KUKA KRL program: MyProgram_270().src

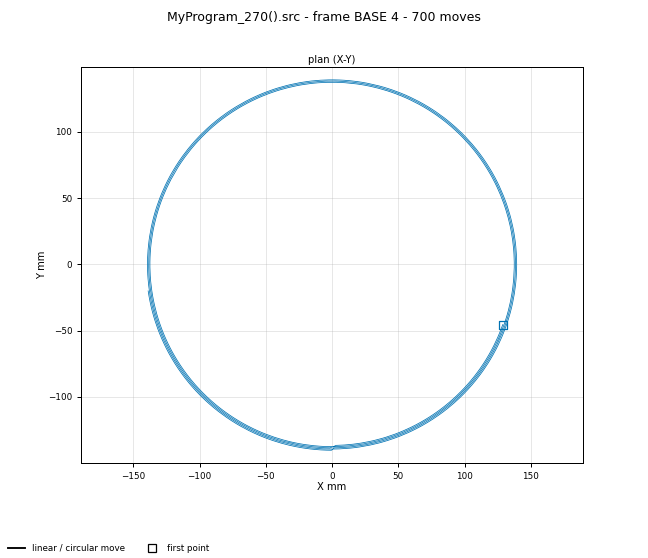
[picture p0: tool path of MyProgram_270().src in frame BASE 4, 700 of 700 moves have a stored position in this frame; points joined in program order, loops and branches not executed]
&ACCESS RVP
&REL 1
&PARAM TEMPLATE = C:\KRC\Roboter\Template\vorgabe
&PARAM EDITMASK = *
DEF MyProgram_270()
; ---- Setting reference (Base) ----
$BASE = BASE_DATA[4]

; --------------------------
; ---- Setting tool (TCP) ----
$TOOL = TOOL_DATA[3]
; --------------------------

$VEL.CP = VEL_APROX_PRINT
Startdeposition()
$VEL.CP = VEL_PRINT
LIN {X 128.8267,Y -45.3786,Z 170,A -18.166,B 9.5893,C 0.2653,E1 9.7435,E2 469.4247} C_DIS
LIN {X 127.6673,Y -48.5446,Z 170,A -19.5524,B 9.5893,C 0.2686,E1 9.7422,E2 470.8092} C_DIS
LIN {X 126.4689,Y -51.5847,Z 170,A -20.9292,B 9.5891,C 0.2724,E1 9.7407,E2 472.1882} C_DIS
LIN {X 125.0288,Y -54.9869,Z 170,A -22.4429,B 9.5891,C 0.2758,E1 9.7391,E2 473.6991} C_DIS
LIN {X 123.6815,Y -57.9517,Z 170,A -23.7911,B 9.589,C 0.2791,E1 9.7375,E2 475.0465} C_DIS
LIN {X 122.1838,Y -61.0461,Z 170,A -25.2077,B 9.5889,C 0.2823,E1 9.7358,E2 476.4613} C_DIS
LIN {X 120.4787,Y -64.3474,Z 170,A -26.8785,B 9.5887,C 0.289,E1 9.7336,E2 478.148} C_DIS
LIN {X 118.4664,Y -67.9811,Z 170,A -28.5284,B 9.5886,C 0.2914,E1 9.7313,E2 479.7881} C_DIS
LIN {X 116.2405,Y -71.7206,Z 170,A -30.2842,B 9.5885,C 0.2944,E1 9.7288,E2 481.5371} C_DIS
LIN {X 114.1692,Y -74.9733,Z 170,A -31.9695,B 9.5883,C 0.3,E1 9.7262,E2 483.2326} C_DIS
LIN {X 111.5417,Y -78.8293,Z 170,A -33.8376,B 9.5883,C 0.3027,E1 9.7233,E2 485.0916} C_DIS
LIN {X 109.2893,Y -81.9245,Z 170,A -35.3836,B 9.5882,C 0.3052,E1 9.7207,E2 486.6318} C_DIS
LIN {X 107.1942,Y -84.647,Z 170,A -36.8457,B 9.588,C 0.3091,E1 9.7182,E2 488.098} C_DIS
LIN {X 104.5097,Y -87.9395,Z 170,A -38.5977,B 9.588,C 0.3125,E1 9.7151,E2 489.8481} C_DIS
LIN {X 102.0952,Y -90.7319,Z 170,A -40.1071,B 9.5878,C 0.3151,E1 9.7123,E2 491.3542} C_DIS
LIN {X 99.655,Y -93.4058,Z 170,A -41.5996,B 9.5878,C 0.3179,E1 9.7095,E2 492.8449} C_DIS
LIN {X 97.2867,Y -95.8696,Z 170,A -43.1095,B 9.5876,C 0.3227,E1 9.7065,E2 494.3659} C_DIS
LIN {X 94.0487,Y -99.0485,Z 170,A -44.8992,B 9.5876,C 0.3241,E1 9.703,E2 496.1433} C_DIS
LIN {X 91.4543,Y -101.4489,Z 170,A -46.374,B 9.5875,C 0.327,E1 9.6999,E2 497.6185} C_DIS
LIN {X 88.8005,Y -103.7798,Z 170,A -47.8905,B 9.5873,C 0.3307,E1 9.6967,E2 499.1409} C_DIS
LIN {X 85.4707,Y -106.5386,Z 170,A -49.6437,B 9.5873,C 0.3328,E1 9.6929,E2 500.8882} C_DIS
LIN {X 82.6267,Y -108.7594,Z 170,A -51.1246,B 9.5872,C 0.3349,E1 9.6896,E2 502.3665} C_DIS
LIN {X 79.7996,Y -110.8504,Z 170,A -52.6158,B 9.5871,C 0.338,E1 9.6863,E2 503.8611} C_DIS
LIN {X 76.3701,Y -113.2397,Z 170,A -54.3449,B 9.587,C 0.3405,E1 9.6823,E2 505.5887} C_DIS
LIN {X 73.3437,Y -115.2233,Z 170,A -55.8332,B 9.587,C 0.3424,E1 9.6788,E2 507.0747} C_DIS
LIN {X 70.377,Y -117.0589,Z 170,A -57.2831,B 9.5868,C 0.3444,E1 9.6754,E2 508.5243} C_DIS
LIN {X 67.0538,Y -118.9933,Z 170,A -58.9763,B 9.5867,C 0.3487,E1 9.6712,E2 510.229} C_DIS
LIN {X 63.1615,Y -121.1024,Z 170,A -60.7503,B 9.5867,C 0.3496,E1 9.6669,E2 511.994} C_DIS
LIN {X 59.6528,Y -122.8711,Z 170,A -62.3575,B 9.5867,C 0.351,E1 9.6629,E2 513.5976} C_DIS
LIN {X 56.5477,Y -124.3307,Z 170,A -63.7852,B 9.5866,C 0.3527,E1 9.6593,E2 515.025} C_DIS
LIN {X 53.8192,Y -125.5337,Z 170,A -65.022,B 9.5866,C 0.3539,E1 9.6561,E2 516.2609} C_DIS
LIN {X 50.4299,Y -126.9344,Z 170,A -66.5584,B 9.5864,C 0.3557,E1 9.6521,E2 517.7984} C_DIS
LIN {X 47.1173,Y -128.2019,Z 170,A -68.0301,B 9.5864,C 0.3571,E1 9.6483,E2 519.2693} C_DIS
LIN {X 43.9464,Y -129.3232,Z 170,A -69.4316,B 9.5864,C 0.3584,E1 9.6446,E2 520.6707} C_DIS
LIN {X 40.9221,Y -130.3108,Z 170,A -70.7407,B 9.5864,C 0.3592,E1 9.6411,E2 521.9775} C_DIS
LIN {X 37.7424,Y -131.267,Z 170,A -72.1466,B 9.5863,C 0.3608,E1 9.6373,E2 523.3861} C_DIS
LIN {X 34.3963,Y -132.1842,Z 170,A -73.588,B 9.5863,C 0.3617,E1 9.6334,E2 524.8268} C_DIS
LIN {X 31.6889,Y -132.8572,Z 170,A -74.7716,B 9.5862,C 0.363,E1 9.6302,E2 526.0128} C_DIS
LIN {X 28.5021,Y -133.5771,Z 170,A -76.1439,B 9.5862,C 0.364,E1 9.6265,E2 527.3863} C_DIS
LIN {X 24.8536,Y -134.3059,Z 170,A -77.6673,B 9.5862,C 0.3643,E1 9.6223,E2 528.906} C_DIS
LIN {X 21.8419,Y -134.8276,Z 170,A -78.9427,B 9.5861,C 0.3649,E1 9.6188,E2 530.1813} C_DIS
LIN {X 18.6875,Y -135.3009,Z 170,A -80.275,B 9.5861,C 0.3655,E1 9.6151,E2 531.5137} C_DIS
LIN {X 15.9333,Y -135.6516,Z 170,A -81.4857,B 9.5861,C 0.367,E1 9.6117,E2 532.7309} C_DIS
LIN {X 12.4247,Y -136.0191,Z 170,A -82.9083,B 9.5861,C 0.3664,E1 9.6078,E2 534.1471} C_DIS
LIN {X 9.1702,Y -136.278,Z 170,A -84.2729,B 9.5861,C 0.3668,E1 9.604,E2 535.5119} C_DIS
LIN {X 6.089,Y -136.4504,Z 170,A -85.5634,B 9.5861,C 0.3671,E1 9.6004,E2 536.8026} C_DIS
LIN {X 3.0317,Y -136.5525,Z 170,A -86.8425,B 9.5861,C 0.3672,E1 9.5968,E2 538.0818} C_DIS
LIN {X 3.0317,Y -136.5525,Z 170,A -86.8425,B 9.5861,C 0.3672,E1 9.5968,E2 538.0818} C_DIS
Enddeposition()
LIN {X 0.9945,Y -137.4915,Z 170,A -87.085,B 9.5192,C 0.3619,E1 9.5293,E2 538.3005} C_DIS
Startdeposition()
$VEL.CP = VEL_PRINT
LIN {X 4.4577,Y -137.425,Z 170,A -85.4345,B 9.5194,C 0.3572,E1 9.534,E2 536.6227} C_DIS
LIN {X 8.6389,Y -137.2242,Z 170,A -83.302,B 9.5198,C 0.3482,E1 9.5401,E2 534.4389} C_DIS
LIN {X 13.382,Y -136.8431,Z 170,A -81.8432,B 9.5194,C 0.3589,E1 9.5439,E2 533.0469} C_DIS
LIN {X 19.4211,Y -136.1171,Z 170,A -79.3116,B 9.5194,C 0.3577,E1 9.5509,E2 530.5142} C_DIS
LIN {X 23.2629,Y -135.5149,Z 170,A -77.6681,B 9.5194,C 0.3562,E1 9.5555,E2 528.8668} C_DIS
LIN {X 27.2986,Y -134.7584,Z 170,A -76.0431,B 9.5194,C 0.3569,E1 9.5599,E2 527.2517} C_DIS
LIN {X 30.5689,Y -134.0543,Z 170,A -74.6502,B 9.5194,C 0.3559,E1 9.5637,E2 525.8579} C_DIS
LIN {X 34.5877,Y -133.0763,Z 170,A -72.9496,B 9.5195,C 0.355,E1 9.5683,E2 524.1592} C_DIS
LIN {X 38.9693,Y -131.8579,Z 170,A -71.0112,B 9.5196,C 0.3523,E1 9.5735,E2 522.2138} C_DIS
LIN {X 45.6098,Y -129.7115,Z 170,A -68.1707,B 9.5196,C 0.3508,E1 9.5811,E2 519.3799} C_DIS
LIN {X 50.1018,Y -128.0424,Z 170,A -66.1842,B 9.5197,C 0.3488,E1 9.5862,E2 517.3932} C_DIS
LIN {X 53.7419,Y -126.56,Z 170,A -64.1199,B 9.5201,C 0.3371,E1 9.5917,E2 515.2725} C_DIS
LIN {X 57.296,Y -124.9893,Z 170,A -63.0785,B 9.5198,C 0.3481,E1 9.5942,E2 514.3044} C_DIS
LIN {X 59.6774,Y -123.8699,Z 170,A -61.8597,B 9.5199,C 0.3438,E1 9.5973,E2 513.0689} C_DIS
LIN {X 62.703,Y -122.3658,Z 170,A -60.4224,B 9.52,C 0.3411,E1 9.6009,E2 511.6267} C_DIS
LIN {X 66.3461,Y -120.4316,Z 170,A -58.5872,B 9.5202,C 0.3359,E1 9.6054,E2 509.7749} C_DIS
LIN {X 70.6496,Y -117.9585,Z 170,A -56.733,B 9.5202,C 0.3376,E1 9.6098,E2 507.9465} C_DIS
LIN {X 72.7662,Y -116.6644,Z 170,A -55.6329,B 9.5202,C 0.3344,E1 9.6125,E2 506.837} C_DIS
LIN {X 76.2614,Y -114.4102,Z 170,A -53.8574,B 9.5204,C 0.3305,E1 9.6166,E2 505.0544} C_DIS
LIN {X 80.3711,Y -111.5619,Z 170,A -51.3205,B 9.5209,C 0.3162,E1 9.6225,E2 502.4569} C_DIS
LIN {X 84.1974,Y -108.7027,Z 170,A -49.8119,B 9.5206,C 0.3237,E1 9.6257,E2 501.0088} C_DIS
LIN {X 87.6291,Y -105.9558,Z 170,A -47.4584,B 9.5211,C 0.308,E1 9.631,E2 498.5859} C_DIS
LIN {X 91.5947,Y -102.5472,Z 170,A -46.0081,B 9.5207,C 0.3207,E1 9.6338,E2 497.2277} C_DIS
LIN {X 96.5572,Y -97.8895,Z 170,A -43.2267,B 9.5209,C 0.3161,E1 9.6394,E2 494.4507} C_DIS
LIN {X 101.1452,Y -93.1405,Z 170,A -40.3451,B 9.5212,C 0.307,E1 9.645,E2 491.5496} C_DIS
LIN {X 103.3355,Y -90.7051,Z 170,A -38.9793,B 9.5212,C 0.3039,E1 9.6476,E2 490.1823} C_DIS
LIN {X 106.1515,Y -87.3928,Z 170,A -37.1754,B 9.5214,C 0.2999,E1 9.6508,E2 488.3775} C_DIS
LIN {X 109.5395,Y -83.1066,Z 170,A -35.0798,B 9.5214,C 0.2989,E1 9.6543,E2 486.3028} C_DIS
LIN {X 111.5125,Y -80.4397,Z 170,A -33.6162,B 9.5216,C 0.2936,E1 9.6568,E2 484.8273} C_DIS
LIN {X 113.8575,Y -77.0841,Z 170,A -31.9629,B 9.5216,C 0.2906,E1 9.6594,E2 483.179} C_DIS
LIN {X 117.9408,Y -70.6793,Z 170,A -29.0515,B 9.5217,C 0.2888,E1 9.6637,E2 480.2969} C_DIS
LIN {X 120.0387,Y -67.0547,Z 170,A -27.0708,B 9.522,C 0.2786,E1 9.6665,E2 478.2841} C_DIS
LIN {X 122.0959,Y -63.2308,Z 170,A -25.3145,B 9.5221,C 0.2751,E1 9.6687,E2 476.5327} C_DIS
LIN {X 124.9836,Y -57.3082,Z 170,A -22.6476,B 9.5223,C 0.2697,E1 9.672,E2 473.8731} C_DIS
LIN {X 126.4048,Y -54.102,Z 170,A -21.2081,B 9.5223,C 0.2663,E1 9.6736,E2 472.4348} C_DIS
LIN {X 127.992,Y -50.2314,Z 170,A -19.2693,B 9.5226,C 0.2568,E1 9.6756,E2 470.469} C_DIS
LIN {X 129.8776,Y -45.1308,Z 170,A -17.2435,B 9.5226,C 0.2563,E1 9.6775,E2 468.4716} C_DIS
LIN {X 131.0142,Y -41.7167,Z 170,A -15.7755,B 9.5227,C 0.2529,E1 9.6788,E2 467.006} C_DIS
LIN {X 132.121,Y -38.0707,Z 170,A -14.1922,B 9.5228,C 0.2485,E1 9.68,E2 465.4217} C_DIS
LIN {X 133.0849,Y -34.5541,Z 170,A -12.7534,B 9.5229,C 0.2461,E1 9.681,E2 463.9916} C_DIS
LIN {X 133.941,Y -31.065,Z 170,A -11.3472,B 9.5229,C 0.244,E1 9.682,E2 462.5954} C_DIS
LIN {X 134.5739,Y -28.2049,Z 170,A -9.7939,B 9.5232,C 0.2325,E1 9.6829,E2 460.9984} C_DIS
LIN {X 135.7493,Y -21.8581,Z 170,A -7.1388,B 9.5234,C 0.2256,E1 9.6841,E2 458.3449} C_DIS
LIN {X 136.3722,Y -17.5435,Z 170,A -5.5976,B 9.5234,C 0.227,E1 9.6847,E2 456.8371} C_DIS
LIN {X 137.0353,Y -11.2466,Z 170,A -3.001,B 9.5235,C 0.2203,E1 9.6854,E2 454.2432} C_DIS
LIN {X 137.4746,Y -2.4202,Z 170,A 0.3604,B 9.5236,C 0.2174,E1 9.6859,E2 450.9192} C_DIS
LIN {X 137.4858,Y 1.6825,Z 170,A 2.4979,B 9.5239,C 0.2021,E1 9.6859,E2 448.7258} C_DIS
LIN {X 137.2829,Y 7.638,Z 170,A 5.1259,B 9.5242,C 0.1914,E1 9.6855,E2 446.077} C_DIS
LIN {X 137.0196,Y 11.4331,Z 170,A 6.7511,B 9.5242,C 0.1858,E1 9.6851,E2 444.4452} C_DIS
LIN {X 136.6061,Y 15.6289,Z 170,A 7.9732,B 9.5242,C 0.1937,E1 9.6848,E2 443.2897} C_DIS
LIN {X 136.2687,Y 18.3336,Z 170,A 9.3236,B 9.5242,C 0.1852,E1 9.6842,E2 441.911} C_DIS
LIN {X 135.7575,Y 21.8067,Z 170,A 10.5805,B 9.5242,C 0.186,E1 9.6837,E2 440.679} C_DIS
LIN {X 135.2539,Y 24.7321,Z 170,A 11.8194,B 9.5243,C 0.1824,E1 9.6831,E2 439.4387} C_DIS
LIN {X 134.373,Y 29.1363,Z 170,A 13.5842,B 9.5243,C 0.1796,E1 9.6821,E2 437.6859} C_DIS
LIN {X 133.6464,Y 32.3057,Z 170,A 14.9678,B 9.5245,C 0.1751,E1 9.6812,E2 436.2976} C_DIS
LIN {X 132.816,Y 35.5659,Z 170,A 16.385,B 9.5245,C 0.1708,E1 9.6802,E2 434.8773} C_DIS
LIN {X 131.8736,Y 38.9155,Z 170,A 17.7516,B 9.5245,C 0.1688,E1 9.6792,E2 433.52} C_DIS
LIN {X 130.8981,Y 42.0801,Z 170,A 19.18,B 9.5247,C 0.1638,E1 9.678,E2 432.0845} C_DIS
LIN {X 129.6333,Y 45.8355,Z 170,A 21.2102,B 9.5249,C 0.1503,E1 9.6761,E2 430.0051} C_DIS
LIN {X 128.3016,Y 49.435,Z 170,A 22.2113,B 9.5247,C 0.1602,E1 9.6752,E2 429.0785} C_DIS
LIN {X 127.125,Y 52.3889,Z 170,A 23.6027,B 9.5248,C 0.1551,E1 9.6737,E2 427.6778} C_DIS
LIN {X 126.162,Y 54.6637,Z 170,A 24.7189,B 9.5248,C 0.1503,E1 9.6724,E2 426.5499} C_DIS
LIN {X 124.6519,Y 58.0255,Z 170,A 26.237,B 9.5249,C 0.1467,E1 9.6707,E2 425.033} C_DIS
LIN {X 123.119,Y 61.2114,Z 170,A 27.7436,B 9.525,C 0.1421,E1 9.6688,E2 423.5213} C_DIS
LIN {X 120.9378,Y 65.4193,Z 170,A 29.7086,B 9.525,C 0.1373,E1 9.6662,E2 421.5563} C_DIS
LIN {X 118.8946,Y 69.0623,Z 170,A 31.4905,B 9.5252,C 0.132,E1 9.6638,E2 419.7682} C_DIS
LIN {X 116.9053,Y 72.3792,Z 170,A 32.9669,B 9.5252,C 0.1312,E1 9.6616,E2 418.3078} C_DIS
LIN {X 114.6044,Y 75.9704,Z 170,A 34.7336,B 9.5252,C 0.1271,E1 9.6589,E2 416.5416} C_DIS
LIN {X 112.1602,Y 79.5342,Z 170,A 36.5435,B 9.5252,C 0.1227,E1 9.656,E2 414.7295} C_DIS
LIN {X 109.5062,Y 83.1507,Z 170,A 38.4153,B 9.5253,C 0.1183,E1 9.6529,E2 412.8565} C_DIS
LIN {X 106.7022,Y 86.7194,Z 170,A 40.289,B 9.5253,C 0.1145,E1 9.6496,E2 410.9842} C_DIS
LIN {X 103.7598,Y 90.2188,Z 170,A 42.1695,B 9.5254,C 0.1109,E1 9.6462,E2 409.106} C_DIS
LIN {X 99.0767,Y 95.3387,Z 170,A 44.8966,B 9.5254,C 0.1086,E1 9.6411,E2 406.3984} C_DIS
LIN {X 96.5488,Y 97.8977,Z 170,A 46.6566,B 9.5255,C 0.0996,E1 9.6375,E2 404.6051} C_DIS
LIN {X 93.4602,Y 100.8503,Z 170,A 48.2466,B 9.5255,C 0.1005,E1 9.6344,E2 403.0385} C_DIS
LIN {X 90.203,Y 103.7736,Z 170,A 50.0397,B 9.5255,C 0.0977,E1 9.6306,E2 401.2487} C_DIS
LIN {X 86.7906,Y 106.644,Z 170,A 51.8616,B 9.5255,C 0.0951,E1 9.6267,E2 399.4308} C_DIS
LIN {X 83.3506,Y 109.3536,Z 170,A 53.6942,B 9.5256,C 0.0918,E1 9.6226,E2 397.5968} C_DIS
LIN {X 78.9782,Y 112.5524,Z 170,A 55.7465,B 9.5256,C 0.0926,E1 9.6181,E2 395.5697} C_DIS
LIN {X 76.5732,Y 114.202,Z 170,A 57.1185,B 9.5256,C 0.0871,E1 9.6148,E2 394.178} C_DIS
LIN {X 72.947,Y 116.5519,Z 170,A 58.917,B 9.5256,C 0.0844,E1 9.6106,E2 392.3796} C_DIS
LIN {X 69.2198,Y 118.8034,Z 170,A 60.7573,B 9.5257,C 0.0812,E1 9.6062,E2 390.5359} C_DIS
LIN {X 65.4765,Y 120.907,Z 170,A 62.5302,B 9.5257,C 0.0791,E1 9.6018,E2 388.7649} C_DIS
LIN {X 60.8601,Y 123.2922,Z 170,A 64.3876,B 9.5257,C 0.0831,E1 9.5973,E2 386.9457} C_DIS
LIN {X 58.71,Y 124.332,Z 170,A 65.5408,B 9.5257,C 0.0784,E1 9.5944,E2 385.773} C_DIS
LIN {X 55.751,Y 125.6859,Z 170,A 66.8596,B 9.5257,C 0.0777,E1 9.591,E2 384.4588} C_DIS
LIN {X 52.3572,Y 127.1383,Z 170,A 68.4709,B 9.5257,C 0.0744,E1 9.5868,E2 382.8386} C_DIS
LIN {X 47.9866,Y 128.8499,Z 170,A 70.365,B 9.5257,C 0.0737,E1 9.5819,E2 380.9522} C_DIS
LIN {X 44.9262,Y 129.9485,Z 170,A 71.7246,B 9.5257,C 0.0724,E1 9.5783,E2 379.5922} C_DIS
LIN {X 41.4522,Y 131.0986,Z 170,A 73.2785,B 9.5258,C 0.0704,E1 9.5742,E2 378.0349} C_DIS
LIN {X 38.1638,Y 132.0937,Z 170,A 74.639,B 9.5258,C 0.0708,E1 9.5706,E2 376.6835} C_DIS
LIN {X 34.9179,Y 132.9888,Z 170,A 76.1705,B 9.5258,C 0.0671,E1 9.5664,E2 375.1363} C_DIS
LIN {X 29.0493,Y 134.3918,Z 170,A 78.6429,B 9.5258,C 0.0664,E1 9.5597,E2 372.6698} C_DIS
LIN {X 25.6384,Y 135.0841,Z 170,A 80.0199,B 9.5258,C 0.0672,E1 9.5559,E2 371.3023} C_DIS
LIN {X 21.8795,Y 135.7457,Z 170,A 81.9193,B 9.5258,C 0.06,E1 9.5506,E2 369.3651} C_DIS
LIN {X 18.5277,Y 136.2432,Z 170,A 83.1255,B 9.5258,C 0.0638,E1 9.5473,E2 368.1849} C_DIS
LIN {X 9.7314,Y 137.1512,Z 170,A 87.6017,B 9.5259,C 0.0464,E1 9.5346,E2 363.6113} C_DIS
LIN {X 3.0399,Y 137.4642,Z 170,A 89.441,B 9.5259,C 0.066,E1 9.5298,E2 361.892} C_DIS
LIN {X -4.0559,Y 137.4362,Z 170,A 92.5213,B 9.5259,C 0.0637,E1 9.5212,E2 358.798} C_DIS
LIN {X -10.5289,Y 137.093,Z 170,A 95.0095,B 9.5259,C 0.0686,E1 9.5143,E2 356.3376} C_DIS
LIN {X -15.8028,Y 136.5853,Z 170,A 97.2212,B 9.5259,C 0.0692,E1 9.5082,E2 354.1268} C_DIS
LIN {X -19.7314,Y 136.0727,Z 170,A 99.2909,B 9.5259,C 0.0615,E1 9.5023,E2 352.0062} C_DIS
LIN {X -22.8961,Y 135.5761,Z 170,A 100.445,B 9.5259,C 0.0658,E1 9.4992,E2 350.8753} C_DIS
LIN {X -26.4326,Y 134.9321,Z 170,A 101.8121,B 9.5259,C 0.0693,E1 9.4955,E2 349.5254} C_DIS
LIN {X -30.0751,Y 134.1671,Z 170,A 103.299,B 9.5258,C 0.0715,E1 9.4915,E2 348.0474} C_DIS
LIN {X -32.9598,Y 133.4887,Z 170,A 104.7956,B 9.5258,C 0.0672,E1 9.4873,E2 346.5193} C_DIS
LIN {X -36.4161,Y 132.5868,Z 170,A 106.0641,B 9.5258,C 0.0727,E1 9.484,E2 345.279} C_DIS
LIN {X -38.7478,Y 131.9227,Z 170,A 107.164,B 9.5258,C 0.0718,E1 9.481,E2 344.1687} C_DIS
LIN {X -42.1894,Y 130.8632,Z 170,A 108.6839,B 9.5258,C 0.0728,E1 9.4769,E2 342.6475} C_DIS
LIN {X -47.4616,Y 129.0465,Z 170,A 110.9834,B 9.5258,C 0.0756,E1 9.4709,E2 340.3529} C_DIS
LIN {X -50.5435,Y 127.8707,Z 170,A 112.3743,B 9.5258,C 0.0768,E1 9.4673,E2 338.961} C_DIS
LIN {X -53.0087,Y 126.8662,Z 170,A 113.5509,B 9.5258,C 0.0768,E1 9.4642,E2 337.7768} C_DIS
LIN {X -56.2114,Y 125.48,Z 170,A 115.0568,B 9.5258,C 0.0775,E1 9.4603,E2 336.2658} C_DIS
LIN {X -60.7077,Y 123.3674,Z 170,A 117.1893,B 9.5258,C 0.079,E1 9.455,E2 334.1272} C_DIS
LIN {X -64.1612,Y 121.6073,Z 170,A 118.6667,B 9.5257,C 0.0838,E1 9.4513,E2 332.6682} C_DIS
LIN {X -68.4978,Y 119.2213,Z 170,A 120.6402,B 9.5257,C 0.0885,E1 9.4466,E2 330.7076} C_DIS
LIN {X -71.2735,Y 117.5823,Z 170,A 122.1968,B 9.5257,C 0.0865,E1 9.4428,E2 329.1258} C_DIS
LIN {X -75.2749,Y 115.0623,Z 170,A 124.2278,B 9.5257,C 0.0886,E1 9.438,E2 327.0892} C_DIS
LIN {X -79.0533,Y 112.4994,Z 170,A 126.2354,B 9.5257,C 0.0898,E1 9.4334,E2 325.0703} C_DIS
LIN {X -83.2571,Y 109.4251,Z 170,A 128.2742,B 9.5256,C 0.0961,E1 9.4288,E2 323.0499} C_DIS
LIN {X -86.4518,Y 106.9187,Z 170,A 129.9768,B 9.5256,C 0.099,E1 9.4251,E2 321.3476} C_DIS
LIN {X -89.6565,Y 104.2459,Z 170,A 131.7422,B 9.5256,C 0.1019,E1 9.4213,E2 319.5806} C_DIS
LIN {X -92.8554,Y 101.4072,Z 170,A 133.4744,B 9.5255,C 0.1063,E1 9.4178,E2 317.8564} C_DIS
LIN {X -95.5595,Y 98.863,Z 170,A 135.0932,B 9.5255,C 0.1081,E1 9.4145,E2 316.2302} C_DIS
LIN {X -98.3091,Y 96.1293,Z 170,A 136.7566,B 9.5255,C 0.1107,E1 9.4112,E2 314.5624} C_DIS
LIN {X -101.2224,Y 93.0564,Z 170,A 138.6214,B 9.5255,C 0.1126,E1 9.4076,E2 312.6871} C_DIS
LIN {X -103.3595,Y 90.6776,Z 170,A 139.946,B 9.5254,C 0.1157,E1 9.4052,E2 311.3648} C_DIS
LIN {X -106.3015,Y 87.2098,Z 170,A 141.8287,B 9.5254,C 0.1202,E1 9.4018,E2 309.4856} C_DIS
LIN {X -111.1312,Y 80.9657,Z 170,A 144.8669,B 9.5251,C 0.1325,E1 9.3968,E2 306.4821} C_DIS
LIN {X -113.9701,Y 76.9178,Z 170,A 147.1856,B 9.5251,C 0.1328,E1 9.393,E2 304.1336} C_DIS
LIN {X -116.37,Y 73.2362,Z 170,A 149.0296,B 9.5251,C 0.1372,E1 9.3902,E2 302.2899} C_DIS
LIN {X -121.6392,Y 64.1005,Z 170,A 153.401,B 9.5249,C 0.1489,E1 9.3842,E2 297.9264} C_DIS
LIN {X -123.7278,Y 59.9749,Z 170,A 155.388,B 9.5249,C 0.1529,E1 9.3817,E2 295.9342} C_DIS
LIN {X -124.9211,Y 57.4434,Z 170,A 156.6945,B 9.5249,C 0.1535,E1 9.3802,E2 294.6114} C_DIS
LIN {X -126.3995,Y 54.1143,Z 170,A 158.1252,B 9.5247,C 0.1591,E1 9.3786,E2 293.1931} C_DIS
LIN {X -127.5661,Y 51.3015,Z 170,A 159.4457,B 9.5247,C 0.1616,E1 9.3772,E2 291.8676} C_DIS
LIN {X -129.0726,Y 47.3905,Z 170,A 161.1772,B 9.5247,C 0.1667,E1 9.3755,E2 290.1398} C_DIS
LIN {X -130.2574,Y 44.0268,Z 170,A 162.6196,B 9.5245,C 0.1716,E1 9.3742,E2 288.7044} C_DIS
LIN {X -131.5575,Y 39.9709,Z 170,A 164.5117,B 9.5245,C 0.1745,E1 9.3726,E2 286.7995} C_DIS
LIN {X -132.4463,Y 36.9185,Z 170,A 165.9239,B 9.5245,C 0.1767,E1 9.3715,E2 285.3779} C_DIS
LIN {X -133.3806,Y 33.3888,Z 170,A 167.3329,B 9.5243,C 0.183,E1 9.3705,E2 283.9845} C_DIS
LIN {X -134.0208,Y 30.7156,Z 170,A 168.5671,B 9.5243,C 0.1847,E1 9.3697,E2 282.7405} C_DIS
LIN {X -134.8923,Y 26.6394,Z 170,A 170.3575,B 9.5243,C 0.1887,E1 9.3687,E2 280.9452} C_DIS
LIN {X -135.5174,Y 23.248,Z 170,A 171.8243,B 9.5241,C 0.1923,E1 9.368,E2 279.4762} C_DIS
LIN {X -136.0982,Y 19.5534,Z 170,A 173.3856,B 9.5241,C 0.1968,E1 9.3674,E2 277.916} C_DIS
LIN {X -136.5238,Y 16.3188,Z 170,A 174.7567,B 9.524,C 0.2005,E1 9.3669,E2 276.5449} C_DIS
LIN {X -136.8808,Y 12.9892,Z 170,A 176.1716,B 9.5239,C 0.2042,E1 9.3665,E2 275.1289} C_DIS
LIN {X -137.2091,Y 8.8831,Z 170,A 177.7682,B 9.5237,C 0.2113,E1 9.3662,E2 273.549} C_DIS
LIN {X -137.3913,Y 5.3579,Z 170,A 179.3949,B 9.5237,C 0.2128,E1 9.366,E2 271.9043} C_DIS
LIN {X -137.482,Y 1.9762,Z 170,A -179.08,B 9.5237,C 0.2149,E1 9.3659,E2 270.3662} C_DIS
LIN {X -137.4795,Y -2.1219,Z 170,A -177.4283,B 9.5235,C 0.2209,E1 9.3659,E2 268.7231} C_DIS
LIN {X -137.3696,Y -5.9157,Z 170,A -175.8673,B 9.5235,C 0.2258,E1 9.3661,E2 267.1662} C_DIS
LIN {X -137.2262,Y -8.6058,Z 170,A -174.6341,B 9.5234,C 0.2271,E1 9.3663,E2 265.9202} C_DIS
LIN {X -136.8748,Y -13.052,Z 170,A -172.7079,B 9.5233,C 0.2313,E1 9.3667,E2 263.9872} C_DIS
LIN {X -136.4996,Y -16.522,Z 170,A -171.3229,B 9.5231,C 0.2367,E1 9.3672,E2 262.6122} C_DIS
LIN {X -136.0747,Y -19.7178,Z 170,A -169.9579,B 9.5231,C 0.2402,E1 9.3677,E2 261.2457} C_DIS
LIN {X -135.4849,Y -23.4416,Z 170,A -168.2186,B 9.5231,C 0.2417,E1 9.3685,E2 259.4867} C_DIS
LIN {X -134.7752,Y -27.216,Z 170,A -166.6955,B 9.5229,C 0.2476,E1 9.3693,E2 257.9745} C_DIS
LIN {X -134.0398,Y -30.6324,Z 170,A -165.235,B 9.5228,C 0.2517,E1 9.3702,E2 256.5148} C_DIS
LIN {X -133.1493,Y -34.3001,Z 170,A -163.6937,B 9.5226,C 0.2566,E1 9.3712,E2 254.9787} C_DIS
LIN {X -132.3595,Y -37.2291,Z 170,A -162.2911,B 9.5226,C 0.2577,E1 9.3723,E2 253.5597} C_DIS
LIN {X -131.2538,Y -40.9634,Z 170,A -160.726,B 9.5225,C 0.2632,E1 9.3736,E2 252.0032} C_DIS
LIN {X -129.8952,Y -45.08,Z 170,A -158.8582,B 9.5224,C 0.267,E1 9.3752,E2 250.129} C_DIS
LIN {X -128.504,Y -48.9102,Z 170,A -157.1902,B 9.5222,C 0.2722,E1 9.3769,E2 248.4662} C_DIS
LIN {X -127.2161,Y -52.17,Z 170,A -155.6848,B 9.5222,C 0.2752,E1 9.3784,E2 246.9562} C_DIS
LIN {X -125.7598,Y -55.5857,Z 170,A -154.0067,B 9.5221,C 0.2769,E1 9.3803,E2 245.2626} C_DIS
LIN {X -123.9324,Y -59.5466,Z 170,A -152.256,B 9.5219,C 0.2829,E1 9.3824,E2 243.5215} C_DIS
LIN {X -122.2336,Y -62.9628,Z 170,A -150.3668,B 9.5219,C 0.2815,E1 9.3848,E2 241.5954} C_DIS
LIN {X -120.688,Y -65.8779,Z 170,A -149.2799,B 9.5217,C 0.2902,E1 9.3862,E2 240.546} C_DIS
LIN {X -118.8524,Y -69.1352,Z 170,A -147.6358,B 9.5217,C 0.2925,E1 9.3885,E2 238.8919} C_DIS
LIN {X -116.6312,Y -72.8195,Z 170,A -145.7881,B 9.5215,C 0.2958,E1 9.3912,E2 237.0382} C_DIS
LIN {X -114.3309,Y -76.3802,Z 170,A -144.0133,B 9.5214,C 0.2999,E1 9.3939,E2 235.2634} C_DIS
LIN {X -111.8192,Y -80.0122,Z 170,A -142.1297,B 9.5213,C 0.3033,E1 9.397,E2 233.3753} C_DIS
LIN {X -109.0791,Y -83.7095,Z 170,A -140.2054,B 9.5211,C 0.3075,E1 9.4002,E2 231.451} C_DIS
LIN {X -106.4299,Y -87.0526,Z 170,A -138.388,B 9.5211,C 0.3107,E1 9.4034,E2 229.6293} C_DIS
LIN {X -103.4688,Y -90.5523,Z 170,A -136.3488,B 9.521,C 0.3124,E1 9.4072,E2 227.5745} C_DIS
LIN {X -100.3268,Y -94.0223,Z 170,A -134.5451,B 9.5208,C 0.3192,E1 9.4105,E2 225.7903} C_DIS
LIN {X -97.7001,Y -96.7482,Z 170,A -132.8483,B 9.5208,C 0.3201,E1 9.4139,E2 224.0789} C_DIS
LIN {X -94.4521,Y -99.9215,Z 170,A -130.9458,B 9.5206,C 0.3235,E1 9.4177,E2 222.1757} C_DIS
LIN {X -90.9651,Y -103.106,Z 170,A -128.9874,B 9.5205,C 0.3274,E1 9.4218,E2 220.2191} C_DIS
LIN {X -87.7266,Y -105.8751,Z 170,A -127.2086,B 9.5204,C 0.3305,E1 9.4256,E2 218.4404} C_DIS
LIN {X -84.36,Y -108.5767,Z 170,A -125.2622,B 9.5204,C 0.3307,E1 9.4299,E2 216.4755} C_DIS
LIN {X -81.0752,Y -111.0515,Z 170,A -123.6739,B 9.5202,C 0.336,E1 9.4334,E2 214.9036} C_DIS
LIN {X -77.7691,Y -113.3907,Z 170,A -121.9819,B 9.5201,C 0.3385,E1 9.4373,E2 213.2113} C_DIS
LIN {X -74.4148,Y -115.6202,Z 170,A -120.2638,B 9.5201,C 0.3403,E1 9.4413,E2 211.4883} C_DIS
LIN {X -70.7525,Y -117.8972,Z 170,A -118.4293,B 9.52,C 0.3421,E1 9.4457,E2 209.6492} C_DIS
LIN {X -66.9621,Y -120.0905,Z 170,A -116.3461,B 9.52,C 0.3394,E1 9.4509,E2 207.5331} C_DIS
LIN {X -63.9984,Y -121.6928,Z 170,A -115.5673,B 9.5196,C 0.3535,E1 9.4526,E2 206.8342} C_DIS
LIN {X -59.6408,Y -123.8874,Z 170,A -113.2186,B 9.5196,C 0.3497,E1 9.4586,E2 204.4453} C_DIS
LIN {X -56.2599,Y -125.4583,Z 170,A -111.5743,B 9.5197,C 0.3496,E1 9.4628,E2 202.7893} C_DIS
LIN {X -52.8618,Y -126.9275,Z 170,A -110.1181,B 9.5196,C 0.3529,E1 9.4665,E2 201.3441} C_DIS
LIN {X -49.5945,Y -128.2396,Z 170,A -108.6646,B 9.5196,C 0.3546,E1 9.4702,E2 199.8922} C_DIS
LIN {X -46.4412,Y -129.4149,Z 170,A -107.2398,B 9.5195,C 0.3554,E1 9.474,E2 198.4644} C_DIS
LIN {X -43.3291,Y -130.4897,Z 170,A -105.7994,B 9.5195,C 0.3551,E1 9.4778,E2 197.0151} C_DIS
LIN {X -39.9457,Y -131.5652,Z 170,A -104.3864,B 9.5195,C 0.3576,E1 9.4816,E2 195.6103} C_DIS
LIN {X -37.0143,Y -132.4195,Z 170,A -103.123,B 9.5194,C 0.3586,E1 9.485,E2 194.3478} C_DIS
LIN {X -31.6634,Y -133.8012,Z 170,A -100.7871,B 9.5194,C 0.3593,E1 9.4913,E2 192.0072} C_DIS
LIN {X -28.7412,Y -134.4583,Z 170,A -99.5308,B 9.5194,C 0.3598,E1 9.4947,E2 190.7496} C_DIS
LIN {X -24.7807,Y -135.2452,Z 170,A -97.3901,B 9.5197,C 0.3509,E1 9.5008,E2 188.5493} C_DIS
LIN {X -20.7,Y -135.9289,Z 170,A -96.0036,B 9.5194,C 0.3585,E1 9.5045,E2 187.2059} C_DIS
LIN {X -14.1478,Y -136.767,Z 170,A -93.3807,B 9.5192,C 0.3619,E1 9.5117,E2 184.5988} C_DIS
LIN {X -9.4126,Y -137.1745,Z 170,A -91.4535,B 9.5192,C 0.3632,E1 9.5171,E2 182.6777} C_DIS
LIN {X -6.1433,Y -137.3605,Z 170,A -90.0529,B 9.5192,C 0.3625,E1 9.521,E2 181.2719} C_DIS
LIN {X -2.6113,Y -137.4714,Z 170,A -88.5618,B 9.5192,C 0.362,E1 9.5252,E2 179.7777} C_DIS
LIN {X 0.9945,Y -137.4915,Z 170,A -87.0824,B 9.5192,C 0.3623,E1 9.5293,E2 178.3005} C_DIS
Enddeposition()
LIN {X 0.9945,Y -137.4915,Z 170,A -87.0824,B 9.5192,C 0.3623,E1 9.5293,E2 178.3005} C_DIS
Startdeposition()
$VEL.CP = VEL_PRINT
LIN {X -1.572,Y -138.4006,Z 170,A -88.7848,B 9.4514,C 0.3834,E1 9.4572,E2 180.1395} C_DIS
LIN {X -5.7228,Y -138.2896,Z 170,A -90.3999,B 9.4515,C 0.3813,E1 9.4527,E2 181.742} C_DIS
LIN {X -9.2888,Y -138.0976,Z 170,A -92.0786,B 9.4513,C 0.3854,E1 9.448,E2 183.4471} C_DIS
LIN {X -13.4546,Y -137.7521,Z 170,A -93.6392,B 9.4515,C 0.3816,E1 9.4437,E2 184.9865} C_DIS
LIN {X -20.4329,Y -136.8929,Z 170,A -96.8074,B 9.4513,C 0.3862,E1 9.4348,E2 188.1888} C_DIS
LIN {X -23.6197,Y -136.3791,Z 170,A -98.06,B 9.4513,C 0.384,E1 9.4314,E2 189.4311} C_DIS
LIN {X -27.197,Y -135.7095,Z 170,A -99.4296,B 9.4515,C 0.3805,E1 9.4277,E2 190.7836} C_DIS
LIN {X -36.375,Y -133.5438,Z 170,A -103.2672,B 9.4517,C 0.377,E1 9.4173,E2 194.6138} C_DIS
LIN {X -40.561,Y -132.3305,Z 170,A -105.142,B 9.4517,C 0.3771,E1 9.4123,E2 196.4978} C_DIS
LIN {X -44.0373,Y -131.2149,Z 170,A -106.6082,B 9.4517,C 0.375,E1 9.4084,E2 197.9585} C_DIS
LIN {X -47.1126,Y -130.1421,Z 170,A -107.9691,B 9.4517,C 0.3741,E1 9.4048,E2 199.3212} C_DIS
LIN {X -50.3994,Y -128.9049,Z 170,A -109.4519,B 9.4518,C 0.3734,E1 9.4009,E2 200.8079} C_DIS
LIN {X -54.1672,Y -127.3699,Z 170,A -111.2808,B 9.4518,C 0.3745,E1 9.3962,E2 202.6553} C_DIS
LIN {X -57.5285,Y -125.8863,Z 170,A -112.574,B 9.452,C 0.3684,E1 9.3929,E2 203.9196} C_DIS
LIN {X -60.2563,Y -124.6038,Z 170,A -114.0197,B 9.452,C 0.3709,E1 9.3892,E2 205.3905} C_DIS
LIN {X -67.3011,Y -120.945,Z 170,A -117.0936,B 9.4522,C 0.3626,E1 9.3817,E2 208.4373} C_DIS
LIN {X -70.3258,Y -119.2116,Z 170,A -118.7525,B 9.4522,C 0.3649,E1 9.3776,E2 210.1237} C_DIS
LIN {X -74.1982,Y -116.841,Z 170,A -120.6256,B 9.4522,C 0.362,E1 9.3732,E2 211.9958} C_DIS
LIN {X -77.4441,Y -114.7148,Z 170,A -122.2485,B 9.4523,C 0.3599,E1 9.3694,E2 213.6205} C_DIS
LIN {X -80.9466,Y -112.2712,Z 170,A -124.5079,B 9.4521,C 0.3664,E1 9.3641,E2 215.9418} C_DIS
LIN {X -84.6016,Y -109.543,Z 170,A -125.6532,B 9.4527,C 0.3492,E1 9.3618,E2 216.9927} C_DIS
LIN {X -88.4574,Y -106.4537,Z 170,A -128.0455,B 9.4527,C 0.3522,E1 9.3565,E2 219.4286} C_DIS
LIN {X -91.7931,Y -103.591,Z 170,A -129.8769,B 9.4527,C 0.3491,E1 9.3527,E2 221.261} C_DIS
LIN {X -94.9893,Y -100.6682,Z 170,A -131.6775,B 9.4529,C 0.3459,E1 9.349,E2 223.062} C_DIS
LIN {X -98.5786,Y -97.1567,Z 170,A -133.665,B 9.4531,C 0.3401,E1 9.345,E2 225.0372} C_DIS
LIN {X -101.1495,Y -94.4768,Z 170,A -135.7602,B 9.4528,C 0.3472,E1 9.3409,E2 227.2023} C_DIS
LIN {X -104.1329,Y -91.1781,Z 170,A -137.0172,B 9.4533,C 0.3326,E1 9.3387,E2 228.3848} C_DIS
LIN {X -106.302,Y -88.6403,Z 170,A -138.614,B 9.4533,C 0.3336,E1 9.3358,E2 230.0083} C_DIS
LIN {X -109.0269,Y -85.2658,Z 170,A -140.4097,B 9.4534,C 0.3296,E1 9.3327,E2 231.8031} C_DIS
LIN {X -111.7122,Y -81.716,Z 170,A -142.2931,B 9.4535,C 0.3262,E1 9.3295,E2 233.6908} C_DIS
LIN {X -114.3154,Y -78.0331,Z 170,A -144.1837,B 9.4537,C 0.3223,E1 9.3265,E2 235.5835} C_DIS
LIN {X -116.7745,Y -74.3028,Z 170,A -146.0512,B 9.4538,C 0.3182,E1 9.3237,E2 237.4521} C_DIS
LIN {X -119.1085,Y -70.5011,Z 170,A -147.9709,B 9.4539,C 0.315,E1 9.3209,E2 239.38} C_DIS
LIN {X -121.481,Y -66.3281,Z 170,A -150.0549,B 9.454,C 0.3118,E1 9.318,E2 241.4748} C_DIS
LIN {X -123.4783,Y -62.5274,Z 170,A -151.6631,B 9.4543,C 0.3042,E1 9.316,E2 243.0606} C_DIS
LIN {X -125.0082,Y -59.4098,Z 170,A -153.1227,B 9.4543,C 0.3009,E1 9.3142,E2 244.5221} C_DIS
LIN {X -126.4852,Y -56.1971,Z 170,A -154.5994,B 9.4545,C 0.2973,E1 9.3125,E2 245.9994} C_DIS
LIN {X -128.0705,Y -52.489,Z 170,A -156.5437,B 9.4545,C 0.2978,E1 9.3104,E2 247.9771} C_DIS
LIN {X -129.9848,Y -47.5487,Z 170,A -158.8705,B 9.4545,C 0.2942,E1 9.3081,E2 250.3189} C_DIS
LIN {X -131.1728,Y -44.1638,Z 170,A -159.869,B 9.455,C 0.2816,E1 9.3073,E2 251.2553} C_DIS
LIN {X -132.3782,Y -40.4049,Z 170,A -161.6607,B 9.455,C 0.2799,E1 9.3058,E2 253.0656} C_DIS
LIN {X -133.3619,Y -37.03,Z 170,A -163.1584,B 9.4551,C 0.2766,E1 9.3046,E2 254.5674} C_DIS
LIN {X -134.2491,Y -33.6732,Z 170,A -164.6053,B 9.4552,C 0.2728,E1 9.3036,E2 256.0144} C_DIS
LIN {X -135.1774,Y -29.7308,Z 170,A -166.3798,B 9.4553,C 0.2698,E1 9.3025,E2 257.7998} C_DIS
LIN {X -135.929,Y -26.0747,Z 170,A -167.947,B 9.4554,C 0.2658,E1 9.3016,E2 259.3684} C_DIS
LIN {X -136.5236,Y -22.7571,Z 170,A -169.3043,B 9.4556,C 0.2611,E1 9.301,E2 260.7198} C_DIS
LIN {X -137.0405,Y -19.4042,Z 170,A -170.7518,B 9.4556,C 0.2578,E1 9.3004,E2 262.1714} C_DIS
LIN {X -137.5393,Y -15.4931,Z 170,A -172.6758,B 9.4556,C 0.2582,E1 9.2998,E2 264.1303} C_DIS
LIN {X -137.8636,Y -12.2741,Z 170,A -173.6611,B 9.4559,C 0.2482,E1 9.2995,E2 265.0704} C_DIS
LIN {X -138.1246,Y -8.8517,Z 170,A -175.2752,B 9.4559,C 0.2475,E1 9.2992,E2 266.7072} C_DIS
LIN {X -138.3207,Y -4.9258,Z 170,A -177.1567,B 9.4559,C 0.2471,E1 9.299,E2 268.6188} C_DIS
LIN {X -138.4012,Y -1.4788,Z 170,A -178.6371,B 9.456,C 0.2439,E1 9.299,E2 270.1045} C_DIS
LIN {X -138.3939,Y 1.971,Z 170,A -179.5488,B 9.4563,C 0.2308,E1 9.299,E2 270.9505} C_DIS
LIN {X -138.3242,Y 4.8346,Z 170,A 178.9707,B 9.4563,C 0.2325,E1 9.299,E2 272.4666} C_DIS
LIN {X -138.0025,Y 10.5923,Z 170,A 176.65,B 9.4565,C 0.2244,E1 9.2995,E2 274.7768} C_DIS
LIN {X -137.5562,Y 15.3358,Z 170,A 174.6422,B 9.4566,C 0.2193,E1 9.3,E2 276.787} C_DIS
LIN {X -137.0986,Y 18.9975,Z 170,A 173.0052,B 9.4566,C 0.2168,E1 9.3006,E2 278.4361} C_DIS
LIN {X -136.4498,Y 23.1996,Z 170,A 171.2289,B 9.4568,C 0.212,E1 9.3014,E2 280.2126} C_DIS
LIN {X -135.3082,Y 29.125,Z 170,A 168.7378,B 9.4569,C 0.2047,E1 9.3028,E2 282.7002} C_DIS
LIN {X -134.5581,Y 32.4143,Z 170,A 167.2929,B 9.4569,C 0.2015,E1 9.3037,E2 284.1497} C_DIS
LIN {X -133.674,Y 35.8867,Z 170,A 165.8185,B 9.4571,C 0.1972,E1 9.3047,E2 285.6214} C_DIS
LIN {X -132.7531,Y 39.1566,Z 170,A 164.3862,B 9.4571,C 0.1937,E1 9.3058,E2 287.0556} C_DIS
LIN {X -131.7388,Y 42.4447,Z 170,A 162.9363,B 9.4572,C 0.1902,E1 9.3071,E2 288.5071} C_DIS
LIN {X -130.683,Y 45.5912,Z 170,A 161.5458,B 9.4572,C 0.1866,E1 9.3083,E2 289.8982} C_DIS
LIN {X -129.5782,Y 48.6417,Z 170,A 160.1593,B 9.4574,C 0.1837,E1 9.3097,E2 291.2886} C_DIS
LIN {X -128.236,Y 52.0784,Z 170,A 158.6132,B 9.4574,C 0.1799,E1 9.3113,E2 292.8354} C_DIS
LIN {X -126.7925,Y 55.5028,Z 170,A 157.0987,B 9.4575,C 0.1753,E1 9.3129,E2 294.3454} C_DIS
LIN {X -125.5537,Y 58.2478,Z 170,A 155.7226,B 9.4575,C 0.1742,E1 9.3145,E2 295.7361} C_DIS
LIN {X -124.021,Y 61.4437,Z 170,A 154.2997,B 9.4576,C 0.1696,E1 9.3163,E2 297.152} C_DIS
LIN {X -122.3771,Y 64.6564,Z 170,A 152.7916,B 9.4576,C 0.166,E1 9.3182,E2 298.6603} C_DIS
LIN {X -118.5619,Y 71.4155,Z 170,A 149.7215,B 9.4579,C 0.1553,E1 9.3225,E2 301.7095} C_DIS
LIN {X -116.2032,Y 75.1925,Z 170,A 147.7148,B 9.4579,C 0.1536,E1 9.3255,E2 303.7345} C_DIS
LIN {X -113.9921,Y 78.5042,Z 170,A 145.9137,B 9.4579,C 0.1523,E1 9.3283,E2 305.5527} C_DIS
LIN {X -111.3235,Y 82.2451,Z 170,A 143.8098,B 9.4579,C 0.1513,E1 9.3318,E2 307.6794} C_DIS
LIN {X -108.3636,Y 86.1068,Z 170,A 142.0736,B 9.4581,C 0.1417,E1 9.3347,E2 309.3794} C_DIS
LIN {X -105.9152,Y 89.1013,Z 170,A 140.3248,B 9.4581,C 0.1407,E1 9.3379,E2 311.1446} C_DIS
LIN {X -100.9987,Y 94.6387,Z 170,A 137.1899,B 9.4581,C 0.1353,E1 9.3437,E2 314.2851} C_DIS
LIN {X -97.7556,Y 97.9845,Z 170,A 135.2676,B 9.4582,C 0.1311,E1 9.3475,E2 316.2046} C_DIS
LIN {X -93.6655,Y 101.9011,Z 170,A 132.7597,B 9.4582,C 0.1293,E1 9.3526,E2 318.7302} C_DIS
LIN {X -90.7131,Y 104.5387,Z 170,A 131.2807,B 9.4583,C 0.1232,E1 9.3557,E2 320.1881} C_DIS
LIN {X -87.639,Y 107.1282,Z 170,A 129.6,B 9.4583,C 0.1204,E1 9.3593,E2 321.8693} C_DIS
LIN {X -83.974,Y 110.0247,Z 170,A 127.5793,B 9.4583,C 0.1184,E1 9.3638,E2 323.8988} C_DIS
LIN {X -80.1083,Y 112.871,Z 170,A 125.8662,B 9.4585,C 0.1099,E1 9.3676,E2 325.5763} C_DIS
LIN {X -77.8867,Y 114.4152,Z 170,A 124.4353,B 9.4585,C 0.1138,E1 9.3709,E2 327.0444} C_DIS
LIN {X -73.2024,Y 117.4669,Z 170,A 122.1509,B 9.4585,C 0.1096,E1 9.3763,E2 329.3231} C_DIS
LIN {X -66.7925,Y 121.2267,Z 170,A 119.2546,B 9.4585,C 0.1016,E1 9.3832,E2 332.1947} C_DIS
LIN {X -63.9198,Y 122.7639,Z 170,A 117.6976,B 9.4585,C 0.1037,E1 9.3871,E2 333.7761} C_DIS
LIN {X -58.9045,Y 125.2496,Z 170,A 115.4355,B 9.4586,C 0.0996,E1 9.3928,E2 336.0296} C_DIS
LIN {X -56.1378,Y 126.5117,Z 170,A 114.1897,B 9.4586,C 0.0978,E1 9.396,E2 337.2727} C_DIS
LIN {X -53.3057,Y 127.7302,Z 170,A 112.9106,B 9.4586,C 0.0964,E1 9.3993,E2 338.5511} C_DIS
LIN {X -49.8905,Y 129.1028,Z 170,A 111.2831,B 9.4586,C 0.0967,E1 9.4035,E2 340.1901} C_DIS
LIN {X -44.3861,Y 131.0988,Z 170,A 108.9772,B 9.4586,C 0.092,E1 9.4095,E2 342.4799} C_DIS
LIN {X -40.3631,Y 132.391,Z 170,A 107.133,B 9.4586,C 0.0923,E1 9.4145,E2 344.3344} C_DIS
LIN {X -36.9899,Y 133.3731,Z 170,A 105.738,B 9.4586,C 0.0899,E1 9.4182,E2 345.7211} C_DIS
LIN {X -33.6356,Y 134.2586,Z 170,A 104.256,B 9.4587,C 0.0897,E1 9.4222,E2 347.2077} C_DIS
LIN {X -29.8334,Y 135.1553,Z 170,A 102.5766,B 9.4587,C 0.0898,E1 9.4268,E2 348.8938} C_DIS
LIN {X -26.3181,Y 135.8825,Z 170,A 101.039,B 9.4587,C 0.09,E1 9.431,E2 350.4368} C_DIS
LIN {X -19.3456,Y 137.0489,Z 170,A 98.4359,B 9.4587,C 0.0821,E1 9.4381,E2 352.9984} C_DIS
LIN {X -11.1996,Y 137.9543,Z 170,A 94.9776,B 9.4587,C 0.0823,E1 9.4477,E2 356.4631} C_DIS
LIN {X -4.6273,Y 138.3323,Z 170,A 92.1117,B 9.4587,C 0.0847,E1 9.4558,E2 359.3452} C_DIS
LIN {X -1.0604,Y 138.4038,Z 170,A 90.3122,B 9.4587,C 0.0911,E1 9.4609,E2 361.1835} C_DIS
LIN {X 2.2042,Y 138.3901,Z 170,A 89.2057,B 9.4587,C 0.0861,E1 9.4639,E2 362.2593} C_DIS
LIN {X 9.2303,Y 138.1013,Z 170,A 86.2094,B 9.4587,C 0.0882,E1 9.4723,E2 365.2651} C_DIS
LIN {X 16.963,Y 137.3652,Z 170,A 83.3768,B 9.4587,C 0.0812,E1 9.48,E2 368.0493} C_DIS
LIN {X 22.8962,Y 136.5004,Z 170,A 80.6461,B 9.4587,C 0.0874,E1 9.4877,E2 370.8101} C_DIS
LIN {X 26.7327,Y 135.8032,Z 170,A 78.0684,B 9.4585,C 0.1082,E1 9.4951,E2 373.5051} C_DIS
LIN {X 33.542,Y 134.2824,Z 170,A 76.2884,B 9.4587,C 0.087,E1 9.4995,E2 375.149} C_DIS
LIN {X 37.5398,Y 133.2193,Z 170,A 74.431,B 9.4587,C 0.0913,E1 9.5045,E2 377.0239} C_DIS
LIN {X 40.7774,Y 132.2642,Z 170,A 73.0747,B 9.4587,C 0.0915,E1 9.5082,E2 378.3749} C_DIS
LIN {X 43.8865,Y 131.2651,Z 170,A 71.7099,B 9.4587,C 0.093,E1 9.5118,E2 379.7411} C_DIS
LIN {X 47.2503,Y 130.0924,Z 170,A 70.2267,B 9.4587,C 0.0946,E1 9.5157,E2 381.2252} C_DIS
LIN {X 51.2121,Y 128.5852,Z 170,A 68.2972,B 9.4586,C 0.1001,E1 9.5208,E2 383.1762} C_DIS
LIN {X 55.3635,Y 126.8527,Z 170,A 66.6783,B 9.4586,C 0.097,E1 9.5248,E2 384.765} C_DIS
LIN {X 58.889,Y 125.257,Z 170,A 64.1825,B 9.4584,C 0.1182,E1 9.5314,E2 387.3705} C_DIS
LIN {X 64.6652,Y 122.3725,Z 170,A 62.4048,B 9.4586,C 0.1023,E1 9.5356,E2 389.0384} C_DIS
LIN {X 68.3209,Y 120.3719,Z 170,A 60.5952,B 9.4586,C 0.1065,E1 9.54,E2 390.8586} C_DIS
LIN {X 72.3595,Y 117.9879,Z 170,A 58.83,B 9.4586,C 0.1055,E1 9.5442,E2 392.6022} C_DIS
LIN {X 75.6205,Y 115.9253,Z 170,A 57.0875,B 9.4585,C 0.1112,E1 9.5483,E2 394.3629} C_DIS
LIN {X 81.9386,Y 111.5487,Z 170,A 54.0229,B 9.4585,C 0.1138,E1 9.5553,E2 397.4136} C_DIS
LIN {X 85.1896,Y 109.0868,Z 170,A 52.23,B 9.4584,C 0.1191,E1 9.5593,E2 399.2198} C_DIS
LIN {X 88.7185,Y 106.2364,Z 170,A 50.376,B 9.4584,C 0.122,E1 9.5633,E2 401.0714} C_DIS
LIN {X 92.2502,Y 103.1841,Z 170,A 48.5251,B 9.4584,C 0.1238,E1 9.5671,E2 402.9127} C_DIS
LIN {X 96.9867,Y 98.7453,Z 170,A 46.1076,B 9.4584,C 0.123,E1 9.572,E2 405.2975} C_DIS
LIN {X 102.97,Y 92.4893,Z 170,A 42.5161,B 9.4582,C 0.1307,E1 9.5789,E2 408.8915} C_DIS
LIN {X 105.1536,Y 89.9998,Z 170,A 40.9311,B 9.4582,C 0.1385,E1 9.5818,E2 410.5038} C_DIS
LIN {X 108.0367,Y 86.5175,Z 170,A 39.068,B 9.4581,C 0.1425,E1 9.5851,E2 412.3667} C_DIS
LIN {X 110.8077,Y 82.9387,Z 170,A 37.202,B 9.458,C 0.1466,E1 9.5883,E2 414.2326} C_DIS
LIN {X 113.5703,Y 79.1128,Z 170,A 35.2806,B 9.458,C 0.1504,E1 9.5914,E2 416.151} C_DIS
LIN {X 116.2523,Y 75.1169,Z 170,A 33.3235,B 9.4579,C 0.1544,E1 9.5944,E2 418.1049} C_DIS
LIN {X 119.6087,Y 69.6487,Z 170,A 30.7475,B 9.4578,C 0.1591,E1 9.5981,E2 420.6724} C_DIS
LIN {X 121.6745,Y 65.9734,Z 170,A 28.9675,B 9.4578,C 0.1643,E1 9.6005,E2 422.4578} C_DIS
LIN {X 123.5002,Y 62.4844,Z 170,A 27.4419,B 9.4577,C 0.1661,E1 9.6024,E2 423.9712} C_DIS
LIN {X 125.4102,Y 58.558,Z 170,A 25.8278,B 9.4577,C 0.1662,E1 9.6044,E2 425.5623} C_DIS
LIN {X 126.5876,Y 55.9681,Z 170,A 24.5518,B 9.4576,C 0.1716,E1 9.6058,E2 426.8514} C_DIS
LIN {X 128.5604,Y 51.2736,Z 170,A 22.6725,B 9.4576,C 0.1719,E1 9.6078,E2 428.7034} C_DIS
LIN {X 129.8045,Y 48.0377,Z 170,A 21.0837,B 9.4574,C 0.1794,E1 9.6094,E2 430.3127} C_DIS
LIN {X 130.9108,Y 44.9339,Z 170,A 19.7213,B 9.4574,C 0.1831,E1 9.6107,E2 431.6759} C_DIS
LIN {X 131.9144,Y 41.8947,Z 170,A 18.4046,B 9.4573,C 0.1865,E1 9.6118,E2 432.9926} C_DIS
LIN {X 132.8998,Y 38.6556,Z 170,A 17.0332,B 9.4573,C 0.1897,E1 9.6129,E2 434.3613} C_DIS
LIN {X 133.7962,Y 35.4285,Z 170,A 15.6498,B 9.4572,C 0.1935,E1 9.6139,E2 435.7455} C_DIS
LIN {X 134.6045,Y 32.2215,Z 170,A 14.3036,B 9.4571,C 0.1968,E1 9.6148,E2 437.0898} C_DIS
LIN {X 135.7995,Y 26.7521,Z 170,A 11.9637,B 9.4569,C 0.2039,E1 9.6162,E2 439.4347} C_DIS
LIN {X 136.4972,Y 22.9153,Z 170,A 9.9946,B 9.4567,C 0.2169,E1 9.6171,E2 441.4496} C_DIS
LIN {X 137.1393,Y 18.7069,Z 170,A 7.8881,B 9.4563,C 0.2301,E1 9.6179,E2 443.6007} C_DIS
LIN {X 137.8364,Y 12.5767,Z 170,A 6.2174,B 9.4567,C 0.2166,E1 9.6184,E2 445.1629} C_DIS
LIN {X 138.0853,Y 9.4585,Z 170,A 4.2372,B 9.4562,C 0.2366,E1 9.6188,E2 447.2305} C_DIS
LIN {X 138.347,Y 4.1032,Z 170,A 2.1676,B 9.4562,C 0.2395,E1 9.6189,E2 449.2835} C_DIS
LIN {X 138.4067,Y -0.7145,Z 170,A 0.9959,B 9.4565,C 0.2258,E1 9.6189,E2 450.3532} C_DIS
LIN {X 138.3629,Y -3.5279,Z 170,A -1.0443,B 9.4558,C 0.25,E1 9.6188,E2 452.5051} C_DIS
LIN {X 138.1238,Y -8.8636,Z 170,A -2.4422,B 9.4562,C 0.2371,E1 9.6186,E2 453.8026} C_DIS
LIN {X 137.5125,Y -15.7282,Z 170,A -5.3076,B 9.456,C 0.2457,E1 9.6178,E2 456.6726} C_DIS
LIN {X 136.9758,Y -19.8575,Z 170,A -7.288,B 9.4557,C 0.2568,E1 9.6171,E2 458.6872} C_DIS
LIN {X 136.2963,Y -24.0829,Z 170,A -9.258,B 9.4554,C 0.2667,E1 9.6161,E2 460.6841} C_DIS
LIN {X 135.497,Y -28.2412,Z 170,A -10.5073,B 9.4556,C 0.2597,E1 9.6155,E2 461.8715} C_DIS
LIN {X 134.7723,Y -31.5198,Z 170,A -11.8912,B 9.4555,C 0.2635,E1 9.6146,E2 463.2561} C_DIS
LIN {X 133.9969,Y -34.6668,Z 170,A -13.3461,B 9.4553,C 0.2701,E1 9.6136,E2 464.7268} C_DIS
LIN {X 132.411,Y -40.2979,Z 170,A -15.3874,B 9.4553,C 0.2678,E1 9.6121,E2 466.7221} C_DIS
LIN {X 131.1517,Y -44.2272,Z 170,A -17.2916,B 9.4551,C 0.2773,E1 9.6104,E2 468.6532} C_DIS
LIN {X 129.9867,Y -47.5434,Z 170,A -19.3481,B 9.4545,C 0.2956,E1 9.6084,E2 470.7876} C_DIS
LIN {X 128.1498,Y -52.2923,Z 170,A -20.8034,B 9.4548,C 0.2859,E1 9.6069,E2 472.1625} C_DIS
LIN {X 124.2669,Y -60.9454,Z 170,A -24.4878,B 9.4547,C 0.2908,E1 9.6027,E2 475.8203} C_DIS
LIN {X 123.0226,Y -63.4227,Z 170,A -25.9458,B 9.4544,C 0.3012,E1 9.6008,E2 477.3192} C_DIS
LIN {X 120.7976,Y -67.5653,Z 170,A -27.8265,B 9.4543,C 0.3047,E1 9.5983,E2 479.1936} C_DIS
LIN {X 118.9518,Y -70.7639,Z 170,A -29.3459,B 9.4541,C 0.3084,E1 9.5961,E2 480.7135} C_DIS
LIN {X 115.6538,Y -76.0346,Z 170,A -31.6382,B 9.4541,C 0.3082,E1 9.5928,E2 482.9725} C_DIS
LIN {X 114.0694,Y -78.3915,Z 170,A -33.0399,B 9.4539,C 0.3164,E1 9.5905,E2 484.4044} C_DIS
LIN {X 110.8944,Y -82.8222,Z 170,A -35.8777,B 9.4532,C 0.3354,E1 9.5857,E2 487.3184} C_DIS
LIN {X 107.4236,Y -87.2776,Z 170,A -37.3107,B 9.4538,C 0.3198,E1 9.5834,E2 488.6387} C_DIS
LIN {X 103.0518,Y -92.3979,Z 170,A -40.1078,B 9.4535,C 0.3264,E1 9.5783,E2 491.4401} C_DIS
LIN {X 98.3995,Y -97.3379,Z 170,A -42.8083,B 9.4535,C 0.33,E1 9.5731,E2 494.1296} C_DIS
LIN {X 96.2393,Y -99.4738,Z 170,A -44.6436,B 9.4528,C 0.3461,E1 9.5693,E2 496.0402} C_DIS
LIN {X 93.386,Y -102.1579,Z 170,A -45.8146,B 9.4531,C 0.339,E1 9.567,E2 497.1552} C_DIS
LIN {X 87.8396,Y -106.9643,Z 170,A -48.9089,B 9.4528,C 0.3464,E1 9.5604,E2 500.2598} C_DIS
LIN {X 81.716,Y -111.7122,Z 170,A -52.4791,B 9.4523,C 0.3606,E1 9.5524,E2 503.8794} C_DIS
LIN {X 78.3465,Y -114.1003,Z 170,A -53.5642,B 9.4527,C 0.3494,E1 9.5501,E2 504.8862} C_DIS
LIN {X 75.8741,Y -115.7594,Z 170,A -55.0117,B 9.4525,C 0.3564,E1 9.5466,E2 506.3625} C_DIS
LIN {X 71.4254,Y -118.5559,Z 170,A -57.2435,B 9.4523,C 0.3612,E1 9.5413,E2 508.6035} C_DIS
LIN {X 67.2058,Y -120.9978,Z 170,A -59.0898,B 9.4523,C 0.3604,E1 9.5369,E2 510.4295} C_DIS
LIN {X 63.8979,Y -122.7754,Z 170,A -60.7763,B 9.4521,C 0.3657,E1 9.5327,E2 512.1343} C_DIS
LIN {X 59.9336,Y -124.7579,Z 170,A -62.4995,B 9.4521,C 0.3657,E1 9.5284,E2 513.8448} C_DIS
LIN {X 54.3364,Y -127.2968,Z 170,A -64.9869,B 9.4521,C 0.3678,E1 9.5221,E2 516.327} C_DIS
LIN {X 51.0166,Y -128.664,Z 170,A -66.9083,B 9.4516,C 0.3792,E1 9.5169,E2 518.3052} C_DIS
LIN {X 47.3074,Y -130.0718,Z 170,A -68.1493,B 9.4519,C 0.3722,E1 9.5138,E2 519.4962} C_DIS
LIN {X 43.0098,Y -131.557,Z 170,A -69.9692,B 9.4519,C 0.3728,E1 9.509,E2 521.3095} C_DIS
LIN {X 40.3514,Y -132.3946,Z 170,A -71.127,B 9.4518,C 0.374,E1 9.5059,E2 522.4687} C_DIS
LIN {X 37.0327,Y -133.3611,Z 170,A -72.5859,B 9.4518,C 0.3759,E1 9.502,E2 523.9322} C_DIS
LIN {X 31.2345,Y -134.8375,Z 170,A -74.86,B 9.4518,C 0.3735,E1 9.4959,E2 526.182} C_DIS
LIN {X 26.2532,Y -135.8949,Z 170,A -77.1446,B 9.4516,C 0.3788,E1 9.4896,E2 528.4906} C_DIS
LIN {X 22.0637,Y -136.639,Z 170,A -79.5915,B 9.451,C 0.3946,E1 9.4826,E2 531.0262} C_DIS
LIN {X 16.5559,Y -137.4138,Z 170,A -80.9157,B 9.4518,C 0.3748,E1 9.4793,E2 532.2267} C_DIS
LIN {X 13.1427,Y -137.7821,Z 170,A -82.8565,B 9.4513,C 0.3866,E1 9.4737,E2 534.235} C_DIS
LIN {X 8.5069,Y -138.1458,Z 170,A -84.5218,B 9.4515,C 0.3817,E1 9.4691,E2 535.8682} C_DIS
LIN {X 4.4836,Y -138.3364,Z 170,A -86.2438,B 9.4515,C 0.3832,E1 9.4643,E2 537.5981} C_DIS
LIN {X 1.005,Y -138.402,Z 170,A -87.0839,B 9.4519,C 0.3707,E1 9.4622,E2 538.3615} C_DIS
Enddeposition()
LIN {X 1.005,Y -138.402,Z 170,A -87.0839,B 9.4519,C 0.3707,E1 9.4622,E2 538.3615} C_DIS
Startdeposition()
$VEL.CP = VEL_PRINT
LIN {X 1.4965,Y -139.3132,Z 170,A -86.5174,B 9.2131,C 0.3745,E1 9.2251,E2 537.8514} C_DIS
LIN {X 5.5486,Y -139.2088,Z 170,A -84.9684,B 9.2131,C 0.3766,E1 9.2294,E2 536.3169} C_DIS
LIN {X 11.0611,Y -138.881,Z 170,A -82.8138,B 9.213,C 0.3784,E1 9.2354,E2 534.1765} C_DIS
LIN {X 13.6438,Y -138.6499,Z 170,A -81.7147,B 9.213,C 0.3772,E1 9.2384,E2 533.0725} C_DIS
LIN {X 17.1015,Y -138.2669,Z 170,A -79.8861,B 9.2134,C 0.368,E1 9.2436,E2 531.1908} C_DIS
LIN {X 20.7522,Y -137.7657,Z 170,A -78.5712,B 9.2132,C 0.3715,E1 9.2472,E2 529.9014} C_DIS
LIN {X 28.7418,Y -136.3237,Z 170,A -75.2903,B 9.2132,C 0.3706,E1 9.2562,E2 526.626} C_DIS
LIN {X 35.28,Y -134.7795,Z 170,A -72.7401,B 9.2132,C 0.373,E1 9.263,E2 524.1019} C_DIS
LIN {X 37.8322,Y -134.0843,Z 170,A -71.5805,B 9.2132,C 0.3704,E1 9.2662,E2 522.9321} C_DIS
LIN {X 41.6465,Y -132.9509,Z 170,A -69.2054,B 9.214,C 0.3525,E1 9.2728,E2 520.4585} C_DIS
LIN {X 47.0837,Y -131.1217,Z 170,A -67.8497,B 9.2132,C 0.3722,E1 9.276,E2 519.2331} C_DIS
LIN {X 51.1257,Y -129.6008,Z 170,A -65.7052,B 9.2136,C 0.362,E1 9.2817,E2 517.039} C_DIS
LIN {X 56.9801,Y -127.1338,Z 170,A -63.1706,B 9.2136,C 0.3605,E1 9.2882,E2 514.5125} C_DIS
LIN {X 60.0283,Y -125.7232,Z 170,A -61.8107,B 9.2137,C 0.3591,E1 9.2916,E2 513.1542} C_DIS
LIN {X 63.6926,Y -123.9083,Z 170,A -60.0844,B 9.2139,C 0.3557,E1 9.296,E2 511.4208} C_DIS
LIN {X 67.8817,Y -121.6656,Z 170,A -58.3171,B 9.2139,C 0.357,E1 9.3002,E2 509.6763} C_DIS
LIN {X 72.2004,Y -119.1528,Z 170,A -55.7369,B 9.2144,C 0.3418,E1 9.3066,E2 507.0252} C_DIS
LIN {X 75.9711,Y -116.7847,Z 170,A -54.3257,B 9.2141,C 0.3483,E1 9.3098,E2 505.6676} C_DIS
LIN {X 81.3314,Y -113.1175,Z 170,A -51.6703,B 9.2143,C 0.344,E1 9.3159,E2 503.0118} C_DIS
LIN {X 84.1949,Y -111.0028,Z 170,A -50.3238,B 9.2143,C 0.344,E1 9.3188,E2 501.6793} C_DIS
LIN {X 87.1913,Y -108.665,Z 170,A -48.6926,B 9.2145,C 0.3395,E1 9.3224,E2 500.0377} C_DIS
LIN {X 92.0788,Y -104.5554,Z 170,A -45.9081,B 9.2148,C 0.3306,E1 9.3284,E2 497.2299} C_DIS
LIN {X 95.9966,Y -100.9705,Z 170,A -43.8881,B 9.2148,C 0.3299,E1 9.3325,E2 495.2293} C_DIS
LIN {X 99.3223,Y -97.7006,Z 170,A -41.7105,B 9.2152,C 0.3198,E1 9.3368,E2 493.0156} C_DIS
LIN {X 102.0825,Y -94.8128,Z 170,A -40.276,B 9.2152,C 0.321,E1 9.3395,E2 491.6068} C_DIS
LIN {X 105.4502,Y -91.0524,Z 170,A -38.3437,B 9.2152,C 0.3197,E1 9.343,E2 489.6912} C_DIS
LIN {X 108.2918,Y -87.654,Z 170,A -35.8704,B 9.2158,C 0.3002,E1 9.3475,E2 487.1303} C_DIS
LIN {X 112.0057,Y -82.8563,Z 170,A -34.3429,B 9.2153,C 0.317,E1 9.3499,E2 485.7274} C_DIS
LIN {X 114.4662,Y -79.4216,Z 170,A -32.685,B 9.2153,C 0.3146,E1 9.3526,E2 484.0781} C_DIS
LIN {X 117.565,Y -74.7578,Z 170,A -30.1911,B 9.2157,C 0.3044,E1 9.3564,E2 481.5568} C_DIS
LIN {X 119.1735,Y -72.1661,Z 170,A -28.8614,B 9.2158,C 0.2995,E1 9.3584,E2 480.216} C_DIS
LIN {X 121.4636,Y -68.2414,Z 170,A -27.0221,B 9.216,C 0.2953,E1 9.3609,E2 478.3785} C_DIS
LIN {X 123.7504,Y -64.0023,Z 170,A -25.1596,B 9.216,C 0.293,E1 9.3633,E2 476.5294} C_DIS
LIN {X 125.2968,Y -60.9186,Z 170,A -22.8996,B 9.2168,C 0.2692,E1 9.3663,E2 474.1575} C_DIS
LIN {X 127.9909,Y -55.0285,Z 170,A -21.1455,B 9.2163,C 0.2837,E1 9.3681,E2 472.52} C_DIS
LIN {X 129.2695,Y -51.9534,Z 170,A -19.3403,B 9.2168,C 0.2696,E1 9.37,E2 470.6565} C_DIS
LIN {X 130.8291,Y -47.8953,Z 170,A -18.0943,B 9.2165,C 0.2776,E1 9.3712,E2 469.4794} C_DIS
LIN {X 131.7663,Y -45.2498,Z 170,A -16.8964,B 9.2166,C 0.2733,E1 9.3723,E2 468.2745} C_DIS
LIN {X 132.9005,Y -41.8041,Z 170,A -15.2468,B 9.2169,C 0.2654,E1 9.3737,E2 466.6029} C_DIS
LIN {X 134.3456,Y -36.898,Z 170,A -13.3568,B 9.2169,C 0.2645,E1 9.3751,E2 464.7384} C_DIS
LIN {X 135.4517,Y -32.5981,Z 170,A -11.5509,B 9.217,C 0.2598,E1 9.3763,E2 462.9333} C_DIS
LIN {X 136.2059,Y -29.2873,Z 170,A -9.6788,B 9.2175,C 0.2444,E1 9.3775,E2 460.9978} C_DIS
LIN {X 137.089,Y -24.8294,Z 170,A -8.5445,B 9.2171,C 0.2566,E1 9.378,E2 459.9572} C_DIS
LIN {X 137.5446,Y -22.1779,Z 170,A -7.1136,B 9.2174,C 0.2457,E1 9.3787,E2 458.4831} C_DIS
LIN {X 138.1546,Y -17.9767,Z 170,A -5.5581,B 9.2174,C 0.2452,E1 9.3793,E2 456.9505} C_DIS
LIN {X 138.5271,Y -14.8349,Z 170,A -3.8393,B 9.2178,C 0.2314,E1 9.3798,E2 455.1761} C_DIS
LIN {X 138.9064,Y -10.7341,Z 170,A -2.5046,B 9.2177,C 0.2351,E1 9.3801,E2 453.8865} C_DIS
LIN {X 139.243,Y -4.6717,Z 170,A 0.014,B 9.2179,C 0.2273,E1 9.3804,E2 451.3628} C_DIS
LIN {X 139.3219,Y -0.0771,Z 170,A 2.1182,B 9.2181,C 0.2167,E1 9.3804,E2 449.229} C_DIS
LIN {X 139.2726,Y 3.6183,Z 170,A 3.5199,B 9.2181,C 0.2151,E1 9.3804,E2 447.8412} C_DIS
LIN {X 139.146,Y 6.9459,Z 170,A 4.51,B 9.2181,C 0.2202,E1 9.3802,E2 446.8989} C_DIS
LIN {X 138.9515,Y 10.1158,Z 170,A 5.863,B 9.2181,C 0.2153,E1 9.38,E2 445.5386} C_DIS
LIN {X 138.6566,Y 13.5743,Z 170,A 7.6923,B 9.2185,C 0.2016,E1 9.3795,E2 443.6561} C_DIS
LIN {X 138.1945,Y 17.6721,Z 170,A 8.7837,B 9.2183,C 0.2111,E1 9.3791,E2 442.6413} C_DIS
LIN {X 137.2788,Y 23.7666,Z 170,A 11.3945,B 9.2185,C 0.2021,E1 9.378,E2 440.0187} C_DIS
LIN {X 136.4765,Y 28.0005,Z 170,A 13.4772,B 9.2187,C 0.1896,E1 9.3769,E2 437.8944} C_DIS
LIN {X 135.7499,Y 31.3346,Z 170,A 14.4948,B 9.2187,C 0.1948,E1 9.3763,E2 436.9254} C_DIS
LIN {X 135.0182,Y 34.3491,Z 170,A 15.8194,B 9.2187,C 0.1901,E1 9.3754,E2 435.5936} C_DIS
LIN {X 134.1562,Y 37.5752,Z 170,A 17.1813,B 9.2187,C 0.1865,E1 9.3743,E2 434.232} C_DIS
LIN {X 133.1495,Y 41.0004,Z 170,A 18.618,B 9.2189,C 0.1832,E1 9.3732,E2 432.7982} C_DIS
LIN {X 132.1405,Y 44.1436,Z 170,A 19.9519,B 9.2189,C 0.18,E1 9.372,E2 431.4664} C_DIS
LIN {X 131.0724,Y 47.2204,Z 170,A 21.4093,B 9.219,C 0.1736,E1 9.3707,E2 429.9928} C_DIS
LIN {X 129.391,Y 51.6519,Z 170,A 23.8611,B 9.2193,C 0.1566,E1 9.3681,E2 427.4748} C_DIS
LIN {X 127.2802,Y 56.6527,Z 170,A 25.1733,B 9.2191,C 0.1723,E1 9.3667,E2 426.2795} C_DIS
LIN {X 126.1499,Y 59.13,Z 170,A 26.4818,B 9.2192,C 0.1649,E1 9.3652,E2 424.9461} C_DIS
LIN {X 124.8039,Y 61.9177,Z 170,A 27.7743,B 9.2192,C 0.1612,E1 9.3636,E2 423.6503} C_DIS
LIN {X 122.9087,Y 65.6039,Z 170,A 29.5519,B 9.2194,C 0.1551,E1 9.3613,E2 421.8624} C_DIS
LIN {X 120.6879,Y 69.6043,Z 170,A 31.5512,B 9.2194,C 0.1477,E1 9.3585,E2 419.8469} C_DIS
LIN {X 119.0548,Y 72.3626,Z 170,A 32.7676,B 9.2195,C 0.1468,E1 9.3567,E2 418.6429} C_DIS
LIN {X 116.5566,Y 76.3214,Z 170,A 34.6216,B 9.2195,C 0.1438,E1 9.3539,E2 416.7969} C_DIS
LIN {X 114.1248,Y 79.9122,Z 170,A 36.3484,B 9.2195,C 0.1409,E1 9.3512,E2 415.0764} C_DIS
LIN {X 111.4745,Y 83.5698,Z 170,A 38.1961,B 9.2197,C 0.1368,E1 9.3481,E2 413.2291} C_DIS
LIN {X 108.694,Y 87.1553,Z 170,A 40.0543,B 9.2197,C 0.1328,E1 9.3449,E2 411.3711} C_DIS
LIN {X 105.7081,Y 90.753,Z 170,A 41.934,B 9.2197,C 0.1296,E1 9.3415,E2 409.496} C_DIS
LIN {X 100.6811,Y 96.2995,Z 170,A 44.8956,B 9.2198,C 0.1257,E1 9.336,E2 406.5482} C_DIS
LIN {X 97.7791,Y 99.2452,Z 170,A 46.6766,B 9.2198,C 0.1205,E1 9.3324,E2 404.7564} C_DIS
LIN {X 93.5691,Y 103.2236,Z 170,A 48.8151,B 9.2198,C 0.1213,E1 9.3281,E2 402.6481} C_DIS
LIN {X 90.8884,Y 105.5916,Z 170,A 50.2352,B 9.2198,C 0.1197,E1 9.3252,E2 401.2341} C_DIS
LIN {X 88.3588,Y 107.7175,Z 170,A 51.8213,B 9.22,C 0.1121,E1 9.3217,E2 399.6188} C_DIS
LIN {X 84.7531,Y 110.5767,Z 170,A 53.6823,B 9.22,C 0.1095,E1 9.3176,E2 397.7615} C_DIS
LIN {X 78.7806,Y 114.9081,Z 170,A 56.8498,B 9.2201,C 0.1015,E1 9.3103,E2 394.5765} C_DIS
LIN {X 76.1195,Y 116.6884,Z 170,A 57.8376,B 9.2201,C 0.1067,E1 9.3081,E2 393.6303} C_DIS
LIN {X 73.101,Y 118.6025,Z 170,A 59.4619,B 9.2201,C 0.1011,E1 9.3042,E2 391.9863} C_DIS
LIN {X 69.2053,Y 120.9171,Z 170,A 61.2972,B 9.2201,C 0.099,E1 9.2998,E2 390.1544} C_DIS
LIN {X 65.3194,Y 123.0588,Z 170,A 64.0064,B 9.2203,C 0.0772,E1 9.2929,E2 387.3323} C_DIS
LIN {X 58.8826,Y 126.2647,Z 170,A 66.0917,B 9.2203,C 0.0927,E1 9.2879,E2 385.3584} C_DIS
LIN {X 55.1024,Y 127.959,Z 170,A 67.7754,B 9.2203,C 0.0911,E1 9.2836,E2 383.6773} C_DIS
LIN {X 51.6335,Y 129.3984,Z 170,A 69.1624,B 9.2203,C 0.0929,E1 9.28,E2 382.3103} C_DIS
LIN {X 48.2434,Y 130.701,Z 170,A 70.6463,B 9.2203,C 0.0916,E1 9.2762,E2 380.8278} C_DIS
LIN {X 45.407,Y 131.7119,Z 170,A 71.89,B 9.2203,C 0.0903,E1 9.2729,E2 379.5836} C_DIS
LIN {X 42.2809,Y 132.7482,Z 170,A 73.2557,B 9.2203,C 0.0889,E1 9.2692,E2 378.2166} C_DIS
LIN {X 38.7885,Y 133.8109,Z 170,A 74.7617,B 9.2203,C 0.0876,E1 9.2652,E2 376.7104} C_DIS
LIN {X 35.3206,Y 134.7686,Z 170,A 76.3966,B 9.2203,C 0.0833,E1 9.2607,E2 375.0562} C_DIS
LIN {X 26.5911,Y 136.7586,Z 170,A 79.9278,B 9.2203,C 0.0843,E1 9.2512,E2 371.545} C_DIS
LIN {X 22.8858,Y 137.4265,Z 170,A 81.773,B 9.2203,C 0.0774,E1 9.246,E2 369.6628} C_DIS
LIN {X 19.2429,Y 137.9846,Z 170,A 82.9372,B 9.2203,C 0.0841,E1 9.2429,E2 368.5435} C_DIS
LIN {X 13.5969,Y 138.6544,Z 170,A 85.0637,B 9.2203,C 0.0877,E1 9.2371,E2 366.4444} C_DIS
LIN {X 9.193,Y 139.0171,Z 170,A 87.4845,B 9.2203,C 0.075,E1 9.2301,E2 363.9484} C_DIS
LIN {X 5.4105,Y 139.2142,Z 170,A 88.9104,B 9.2203,C 0.0776,E1 9.2262,E2 362.5398} C_DIS
LIN {X 1.2168,Y 139.3148,Z 170,A 90.4158,B 9.2203,C 0.082,E1 9.2221,E2 361.0629} C_DIS
LIN {X -2.5162,Y 139.2968,Z 170,A 91.9435,B 9.2203,C 0.0823,E1 9.2178,E2 359.5368} C_DIS
LIN {X -8.8225,Y 139.0399,Z 170,A 94.529,B 9.2203,C 0.0829,E1 9.2106,E2 356.9539} C_DIS
LIN {X -15.5192,Y 138.4535,Z 170,A 97.2439,B 9.2203,C 0.0847,E1 9.2031,E2 354.2469} C_DIS
LIN {X -19.069,Y 138.0095,Z 170,A 99.4405,B 9.2203,C 0.071,E1 9.1968,E2 351.9596} C_DIS
LIN {X -24.4243,Y 137.1615,Z 170,A 100.7139,B 9.2203,C 0.091,E1 9.1936,E2 350.808} C_DIS
LIN {X -28.3965,Y 136.3959,Z 170,A 102.6111,B 9.2203,C 0.0874,E1 9.1883,E2 348.8828} C_DIS
LIN {X -31.2943,Y 135.7591,Z 170,A 103.8251,B 9.2203,C 0.0883,E1 9.185,E2 347.6704} C_DIS
LIN {X -34.4336,Y 134.9968,Z 170,A 105.1947,B 9.2203,C 0.0885,E1 9.1813,E2 346.2965} C_DIS
LIN {X -37.8315,Y 134.0845,Z 170,A 106.6569,B 9.2203,C 0.0893,E1 9.1773,E2 344.8334} C_DIS
LIN {X -40.8722,Y 133.1887,Z 170,A 107.9773,B 9.2203,C 0.0901,E1 9.1738,E2 343.5118} C_DIS
LIN {X -44.0203,Y 132.1816,Z 170,A 109.4355,B 9.2203,C 0.0895,E1 9.1699,E2 342.0422} C_DIS
LIN {X -50.1114,Y 129.9951,Z 170,A 112.421,B 9.2203,C 0.0861,E1 9.162,E2 339.0179} C_DIS
LIN {X -53.6949,Y 128.5558,Z 170,A 113.2998,B 9.2201,C 0.1013,E1 9.16,E2 338.2294} C_DIS
LIN {X -58.5906,Y 126.3997,Z 170,A 115.9049,B 9.2201,C 0.0964,E1 9.1532,E2 335.5754} C_DIS
LIN {X -61.8979,Y 124.8137,Z 170,A 117.3649,B 9.2201,C 0.0992,E1 9.1495,E2 334.1227} C_DIS
LIN {X -65.267,Y 123.0863,Z 170,A 118.9623,B 9.2201,C 0.1006,E1 9.1456,E2 332.5216} C_DIS
LIN {X -72.3053,Y 119.0894,Z 170,A 122.1333,B 9.2201,C 0.1085,E1 9.138,E2 329.3735} C_DIS
LIN {X -76.2209,Y 116.6226,Z 170,A 124.2318,B 9.2201,C 0.1079,E1 9.133,E2 327.2523} C_DIS
LIN {X -79.5454,Y 114.3801,Z 170,A 126.0073,B 9.2201,C 0.1084,E1 9.1288,E2 325.4624} C_DIS
LIN {X -84.6908,Y 110.6243,Z 170,A 128.8897,B 9.2201,C 0.1082,E1 9.1223,E2 322.5493} C_DIS
LIN {X -87.6779,Y 108.2725,Z 170,A 130.1183,B 9.2199,C 0.1172,E1 9.1197,E2 321.3644} C_DIS
LIN {X -90.9111,Y 105.572,Z 170,A 132.4012,B 9.22,C 0.1105,E1 9.1147,E2 319.0137} C_DIS
LIN {X -94.4755,Y 102.3949,Z 170,A 134.4281,B 9.22,C 0.1132,E1 9.1106,E2 316.9807} C_DIS
LIN {X -98.0722,Y 98.9553,Z 170,A 135.8357,B 9.2198,C 0.129,E1 9.1079,E2 315.6558} C_DIS
LIN {X -100.5877,Y 96.3972,Z 170,A 137.8832,B 9.2198,C 0.1219,E1 9.1038,E2 313.5377} C_DIS
LIN {X -103.5534,Y 93.2032,Z 170,A 139.247,B 9.2198,C 0.1335,E1 9.1014,E2 312.2298} C_DIS
LIN {X -105.7743,Y 90.6761,Z 170,A 140.6908,B 9.2197,C 0.1355,E1 9.0987,E2 310.7799} C_DIS
LIN {X -108.7012,Y 87.1463,Z 170,A 142.8168,B 9.2197,C 0.1355,E1 9.0949,E2 308.6255} C_DIS
LIN {X -110.7425,Y 84.5363,Z 170,A 143.7677,B 9.2195,C 0.146,E1 9.0934,E2 307.7278} C_DIS
LIN {X -112.7875,Y 81.7879,Z 170,A 145.4038,B 9.2195,C 0.1453,E1 9.0907,E2 306.0646} C_DIS
LIN {X -115.4663,Y 77.9604,Z 170,A 147.3265,B 9.2195,C 0.1499,E1 9.0876,E2 304.1438} C_DIS
LIN {X -118.0854,Y 73.9327,Z 170,A 149.4587,B 9.2195,C 0.152,E1 9.0844,E2 301.9938} C_DIS
LIN {X -121.2173,Y 68.679,Z 170,A 151.8065,B 9.2193,C 0.1614,E1 9.0811,E2 299.6699} C_DIS
LIN {X -122.5402,Y 66.2897,Z 170,A 153.0823,B 9.2193,C 0.1616,E1 9.0794,E2 298.376} C_DIS
LIN {X -124.2802,Y 62.962,Z 170,A 154.5551,B 9.2192,C 0.1668,E1 9.0775,E2 296.9137} C_DIS
LIN {X -126.0205,Y 59.406,Z 170,A 156.3034,B 9.2192,C 0.1691,E1 9.0754,E2 295.152} C_DIS
LIN {X -127.5099,Y 56.1391,Z 170,A 157.679,B 9.219,C 0.1748,E1 9.0738,E2 293.7907} C_DIS
LIN {X -128.6992,Y 53.3516,Z 170,A 158.9831,B 9.219,C 0.1771,E1 9.0724,E2 292.4806} C_DIS
LIN {X -129.9734,Y 50.1674,Z 170,A 160.3914,B 9.219,C 0.181,E1 9.071,E2 291.0741} C_DIS
LIN {X -131.194,Y 46.8833,Z 170,A 161.8284,B 9.2188,C 0.185,E1 9.0696,E2 289.6391} C_DIS
LIN {X -132.2423,Y 43.8378,Z 170,A 163.2282,B 9.2188,C 0.1874,E1 9.0684,E2 288.2311} C_DIS
LIN {X -133.3465,Y 40.3566,Z 170,A 164.7394,B 9.2187,C 0.1914,E1 9.0671,E2 286.7204} C_DIS
LIN {X -134.5146,Y 36.2733,Z 170,A 166.5532,B 9.2187,C 0.1952,E1 9.0658,E2 284.8998} C_DIS
LIN {X -135.5115,Y 32.35,Z 170,A 168.2066,B 9.2185,C 0.2001,E1 9.0647,E2 283.2496} C_DIS
LIN {X -136.5068,Y 27.8512,Z 170,A 170.1307,B 9.2185,C 0.205,E1 9.0635,E2 281.3237} C_DIS
LIN {X -137.248,Y 23.941,Z 170,A 171.6887,B 9.2183,C 0.2111,E1 9.0628,E2 279.7774} C_DIS
LIN {X -137.6989,Y 21.1858,Z 170,A 172.9039,B 9.2183,C 0.2132,E1 9.0622,E2 278.5548} C_DIS
LIN {X -138.163,Y 17.9122,Z 170,A 174.3242,B 9.2182,C 0.2161,E1 9.0617,E2 277.1281} C_DIS
LIN {X -138.8594,Y 11.3169,Z 170,A 176.8734,B 9.2179,C 0.2271,E1 9.061,E2 274.6044} C_DIS
LIN {X -139.2267,Y 5.0902,Z 170,A 179.7986,B 9.2179,C 0.2284,E1 9.0605,E2 271.6361} C_DIS
LIN {X -139.2948,Y -2.6322,Z 170,A -177.0964,B 9.2176,C 0.2388,E1 9.0605,E2 268.5433} C_DIS
LIN {X -139.1146,Y -7.5722,Z 170,A -175.0527,B 9.2175,C 0.2445,E1 9.0608,E2 266.5001} C_DIS
LIN {X -138.8953,Y -10.8865,Z 170,A -173.3532,B 9.2175,C 0.2427,E1 9.0611,E2 264.7594} C_DIS
LIN {X -138.4098,Y -15.9034,Z 170,A -171.6092,B 9.2172,C 0.2544,E1 9.0616,E2 263.0592} C_DIS
LIN {X -137.821,Y -20.3881,Z 170,A -169.5241,B 9.2172,C 0.2558,E1 9.0624,E2 260.947} C_DIS
LIN {X -137.1622,Y -24.4202,Z 170,A -167.9132,B 9.217,C 0.2618,E1 9.0632,E2 259.3464} C_DIS
LIN {X -136.5108,Y -27.8317,Z 170,A -166.4428,B 9.2169,C 0.2651,E1 9.064,E2 257.8718} C_DIS
LIN {X -135.7641,Y -31.2725,Z 170,A -164.9906,B 9.2168,C 0.2691,E1 9.0649,E2 256.4202} C_DIS
LIN {X -134.9277,Y -34.7059,Z 170,A -163.5079,B 9.2167,C 0.2727,E1 9.0659,E2 254.935} C_DIS
LIN {X -134.0768,Y -37.8588,Z 170,A -162.1608,B 9.2166,C 0.2763,E1 9.0669,E2 253.5883} C_DIS
LIN {X -133.1394,Y -41.0333,Z 170,A -160.7338,B 9.2165,C 0.2789,E1 9.068,E2 252.154} C_DIS
LIN {X -131.8405,Y -45.036,Z 170,A -158.4544,B 9.2166,C 0.274,E1 9.0702,E2 249.8053} C_DIS
LIN {X -130.2257,Y -49.5124,Z 170,A -156.6624,B 9.2164,C 0.2821,E1 9.0719,E2 248.036} C_DIS
LIN {X -128.8561,Y -52.9757,Z 170,A -155.5048,B 9.2161,C 0.2929,E1 9.0731,E2 246.9277} C_DIS
LIN {X -127.7078,Y -55.6834,Z 170,A -154.2213,B 9.216,C 0.2947,E1 9.0745,E2 245.6355} C_DIS
LIN {X -126.3247,Y -58.7527,Z 170,A -152.8338,B 9.2159,C 0.2983,E1 9.0761,E2 244.2486} C_DIS
LIN {X -124.7191,Y -62.0896,Z 170,A -151.252,B 9.2158,C 0.3011,E1 9.0781,E2 242.6602} C_DIS
LIN {X -122.147,Y -67.0112,Z 170,A -149.1588,B 9.2155,C 0.3103,E1 9.0808,E2 240.5929} C_DIS
LIN {X -119.6187,Y -71.4258,Z 170,A -146.893,B 9.2155,C 0.3124,E1 9.084,E2 238.306} C_DIS
LIN {X -117.5994,Y -74.7049,Z 170,A -145.1429,B 9.2154,C 0.3132,E1 9.0866,E2 236.5354} C_DIS
LIN {X -115.0896,Y -78.5163,Z 170,A -143.2237,B 9.2153,C 0.3168,E1 9.0896,E2 234.6117} C_DIS
LIN {X -112.472,Y -82.2218,Z 170,A -141.3359,B 9.2151,C 0.3207,E1 9.0927,E2 232.722} C_DIS
LIN {X -109.7181,Y -85.8619,Z 170,A -139.4371,B 9.2151,C 0.3245,E1 9.0959,E2 230.8213} C_DIS
LIN {X -106.938,Y -89.3008,Z 170,A -137.5894,B 9.2149,C 0.3279,E1 9.0992,E2 228.9707} C_DIS
LIN {X -102.3917,Y -94.4781,Z 170,A -134.6657,B 9.2147,C 0.3322,E1 9.1046,E2 226.0364} C_DIS
LIN {X -98.7719,Y -98.2567,Z 170,A -132.5913,B 9.2145,C 0.338,E1 9.1087,E2 223.9728} C_DIS
LIN {X -95.9696,Y -100.9964,Z 170,A -130.9398,B 9.2145,C 0.3403,E1 9.112,E2 222.3167} C_DIS
LIN {X -92.6067,Y -104.0887,Z 170,A -129.0182,B 9.2143,C 0.3431,E1 9.116,E2 220.3902} C_DIS
LIN {X -89.2057,Y -107.0178,Z 170,A -127.1675,B 9.2143,C 0.3463,E1 9.1199,E2 218.5392} C_DIS
LIN {X -85.6673,Y -109.8706,Z 170,A -125.1003,B 9.2143,C 0.3457,E1 9.1245,E2 216.4467} C_DIS
LIN {X -83.0553,Y -111.8574,Z 170,A -123.5822,B 9.2143,C 0.3447,E1 9.128,E2 214.9068} C_DIS
LIN {X -79.6546,Y -114.3041,Z 170,A -122.2,B 9.2139,C 0.3539,E1 9.131,E2 213.5693} C_DIS
LIN {X -75.7971,Y -116.8977,Z 170,A -120.2846,B 9.2139,C 0.3567,E1 9.1355,E2 211.6537} C_DIS
LIN {X -71.8721,Y -119.3513,Z 170,A -118.3791,B 9.2137,C 0.3594,E1 9.14,E2 209.7482} C_DIS
LIN {X -68.266,Y -121.4497,Z 170,A -116.0449,B 9.2141,C 0.3497,E1 9.1459,E2 207.3331} C_DIS
LIN {X -63.5662,Y -123.9726,Z 170,A -114.246,B 9.2137,C 0.3601,E1 9.1503,E2 205.5861} C_DIS
LIN {X -60.6509,Y -125.4257,Z 170,A -113.0728,B 9.2135,C 0.3649,E1 9.1531,E2 204.4346} C_DIS
LIN {X -55.9066,Y -127.6112,Z 170,A -111.0713,B 9.2133,C 0.3701,E1 9.1582,E2 202.4521} C_DIS
LIN {X -51.9473,Y -129.2719,Z 170,A -109.2337,B 9.2133,C 0.3705,E1 9.163,E2 200.605} C_DIS
LIN {X -48.5948,Y -130.5694,Z 170,A -107.7315,B 9.2133,C 0.3714,E1 9.1669,E2 199.0996} C_DIS
LIN {X -45.15,Y -131.8009,Z 170,A -106.2444,B 9.2132,C 0.373,E1 9.1708,E2 197.6146} C_DIS
LIN {X -42.0461,Y -132.8232,Z 170,A -104.8729,B 9.2132,C 0.3735,E1 9.1745,E2 196.2393} C_DIS
LIN {X -38.1695,Y -133.99,Z 170,A -102.9796,B 9.2133,C 0.3701,E1 9.1796,E2 194.3158} C_DIS
LIN {X -28.6353,Y -136.3467,Z 170,A -99.1702,B 9.213,C 0.377,E1 9.1899,E2 190.5357} C_DIS
LIN {X -22.7118,Y -137.4556,Z 170,A -96.6471,B 9.213,C 0.377,E1 9.1969,E2 188.0061} C_DIS
LIN {X -17.4876,Y -138.2186,Z 170,A -94.5526,B 9.213,C 0.3792,E1 9.2026,E2 185.9209} C_DIS
LIN {X -14.3877,Y -138.5753,Z 170,A -93.1696,B 9.213,C 0.3774,E1 9.2065,E2 184.5245} C_DIS
LIN {X -9.8974,Y -138.9675,Z 170,A -91.3632,B 9.213,C 0.3786,E1 9.2115,E2 182.7235} C_DIS
LIN {X -5.9878,Y -139.1917,Z 170,A -89.6548,B 9.213,C 0.3766,E1 9.2163,E2 181.0016} C_DIS
LIN {X -2.2248,Y -139.3016,Z 170,A -88.2246,B 9.213,C 0.379,E1 9.2203,E2 179.5861} C_DIS
LIN {X 1.007,Y -139.3143,Z 170,A -87.4367,B 9.2125,C 0.3901,E1 9.2223,E2 178.8679} C_DIS
Enddeposition()
LIN {X 1.007,Y -139.3143,Z 170,A -87.4367,B 9.2125,C 0.3901,E1 9.2223,E2 178.8679} C_DIS
Startdeposition()
$VEL.CP = VEL_PRINT
LIN {X -0.5203,Y -140.2304,Z 170,A -88.1526,B 9.212,C 0.3976,E1 9.22,E2 179.6305} C_DIS
LIN {X -4.1645,Y -140.1695,Z 170,A -89.5875,B 9.212,C 0.3966,E1 9.216,E2 181.059} C_DIS
LIN {X -8.3177,Y -139.9845,Z 170,A -91.306,B 9.212,C 0.3969,E1 9.2112,E2 182.7809} C_DIS
LIN {X -12.2391,Y -139.6966,Z 170,A -92.9053,B 9.212,C 0.3966,E1 9.2068,E2 184.3798} C_DIS
LIN {X -16.3419,Y -139.2757,Z 170,A -94.6488,B 9.212,C 0.3975,E1 9.2019,E2 186.1316} C_DIS
LIN {X -20.507,Y -138.725,Z 170,A -96.3344,B 9.2121,C 0.3964,E1 9.1973,E2 187.8138} C_DIS
LIN {X -24.2831,Y -138.113,Z 170,A -97.9585,B 9.2121,C 0.3971,E1 9.1928,E2 189.4462} C_DIS
LIN {X -28.3017,Y -137.3456,Z 170,A -99.5494,B 9.2121,C 0.3947,E1 9.1884,E2 191.027} C_DIS
LIN {X -32.2547,Y -136.4723,Z 170,A -101.2955,B 9.2121,C 0.3957,E1 9.1836,E2 192.7856} C_DIS
LIN {X -38.3349,Y -134.8905,Z 170,A -103.7357,B 9.2123,C 0.3915,E1 9.1771,E2 195.2099} C_DIS
LIN {X -41.2496,Y -134.0267,Z 170,A -105.0154,B 9.2123,C 0.3914,E1 9.1737,E2 196.4947} C_DIS
LIN {X -44.5702,Y -132.9594,Z 170,A -106.4831,B 9.2123,C 0.3911,E1 9.1698,E2 197.9681} C_DIS
LIN {X -47.9801,Y -131.7677,Z 170,A -107.9253,B 9.2124,C 0.3891,E1 9.166,E2 199.4061} C_DIS
LIN {X -51.4861,Y -130.439,Z 170,A -109.4661,B 9.2124,C 0.3879,E1 9.162,E2 200.9483} C_DIS
LIN {X -54.9235,Y -129.0296,Z 170,A -110.9832,B 9.2125,C 0.3863,E1 9.158,E2 202.4654} C_DIS
LIN {X -59.3017,Y -127.0754,Z 170,A -112.9691,B 9.2125,C 0.3847,E1 9.153,E2 204.4549} C_DIS
LIN {X -62.861,Y -125.3548,Z 170,A -115.5126,B 9.2119,C 0.4007,E1 9.1464,E2 207.1178} C_DIS
LIN {X -68.8136,Y -122.1878,Z 170,A -117.3799,B 9.2128,C 0.3801,E1 9.1421,E2 208.871} C_DIS
LIN {X -72.2875,Y -120.1657,Z 170,A -119.1448,B 9.2128,C 0.3802,E1 9.1378,E2 210.6517} C_DIS
LIN {X -76.052,Y -117.8193,Z 170,A -120.9586,B 9.2128,C 0.3776,E1 9.1335,E2 212.4654} C_DIS
LIN {X -79.8142,Y -115.3034,Z 170,A -123.775,B 9.2123,C 0.3929,E1 9.1268,E2 215.4053} C_DIS
LIN {X -85.8774,Y -110.8613,Z 170,A -125.7581,B 9.2133,C 0.3675,E1 9.1227,E2 217.2486} C_DIS
LIN {X -88.863,Y -108.4829,Z 170,A -127.4815,B 9.2133,C 0.3678,E1 9.1189,E2 218.9928} C_DIS
LIN {X -92.4283,Y -105.4622,Z 170,A -129.4152,B 9.2133,C 0.3648,E1 9.1148,E2 220.9292} C_DIS
LIN {X -95.6589,Y -102.5405,Z 170,A -131.2059,B 9.2135,C 0.3617,E1 9.1111,E2 222.7208} C_DIS
LIN {X -99.6337,Y -98.683,Z 170,A -133.4379,B 9.2137,C 0.3567,E1 9.1066,E2 224.948} C_DIS
LIN {X -102.8237,Y -95.3548,Z 170,A -135.914,B 9.2134,C 0.3636,E1 9.1018,E2 227.4993} C_DIS
LIN {X -106.1625,Y -91.6226,Z 170,A -137.2116,B 9.2141,C 0.3457,E1 9.0996,E2 228.7002} C_DIS
LIN {X -108.1349,Y -89.2863,Z 170,A -138.7086,B 9.2141,C 0.3475,E1 9.0968,E2 230.2286} C_DIS
LIN {X -110.9259,Y -85.7941,Z 170,A -140.5794,B 9.2141,C 0.3443,E1 9.0936,E2 232.1042} C_DIS
LIN {X -113.7157,Y -82.0608,Z 170,A -142.5079,B 9.2143,C 0.3404,E1 9.0904,E2 234.0349} C_DIS
LIN {X -116.2144,Y -78.4818,Z 170,A -144.3046,B 9.2145,C 0.3364,E1 9.0875,E2 235.8324} C_DIS
LIN {X -118.585,Y -74.8517,Z 170,A -146.1212,B 9.2145,C 0.333,E1 9.0848,E2 237.6538} C_DIS
LIN {X -120.9987,Y -70.8837,Z 170,A -148.0074,B 9.2148,C 0.3282,E1 9.0821,E2 239.5374} C_DIS
LIN {X -123.2305,Y -66.9289,Z 170,A -149.9814,B 9.2148,C 0.3257,E1 9.0794,E2 241.5255} C_DIS
LIN {X -125.0692,Y -63.4219,Z 170,A -151.4929,B 9.2151,C 0.3197,E1 9.0775,E2 243.0223} C_DIS
LIN {X -126.7406,Y -60.0139,Z 170,A -153.0649,B 9.2151,C 0.316,E1 9.0756,E2 244.5961} C_DIS
LIN {X -128.5558,Y -56.0195,Z 170,A -154.8999,B 9.2153,C 0.3121,E1 9.0735,E2 246.4352} C_DIS
LIN {X -130.2445,Y -51.9734,Z 170,A -156.693,B 9.2155,C 0.3074,E1 9.0716,E2 248.2273} C_DIS
LIN {X -131.5795,Y -48.4974,Z 170,A -158.5427,B 9.2155,C 0.309,E1 9.0697,E2 250.1177} C_DIS
LIN {X -132.7314,Y -45.2497,Z 170,A -159.6435,B 9.2157,C 0.2999,E1 9.0688,E2 251.1784} C_DIS
LIN {X -133.6689,Y -42.3951,Z 170,A -160.9005,B 9.2158,C 0.297,E1 9.0677,E2 252.4382} C_DIS
LIN {X -134.6889,Y -39.0345,Z 170,A -162.373,B 9.2159,C 0.2937,E1 9.0665,E2 253.9144} C_DIS
LIN {X -135.6226,Y -35.657,Z 170,A -163.8917,B 9.2159,C 0.2912,E1 9.0654,E2 255.443} C_DIS
LIN {X -136.6549,Y -31.4671,Z 170,A -165.6196,B 9.2162,C 0.2857,E1 9.0643,E2 257.1651} C_DIS
LIN {X -137.4712,Y -27.6843,Z 170,A -167.1857,B 9.2163,C 0.2809,E1 9.0634,E2 258.7279} C_DIS
LIN {X -138.1656,Y -23.989,Z 170,A -168.9071,B 9.2163,C 0.2798,E1 9.0625,E2 260.4715} C_DIS
LIN {X -138.8032,Y -19.9599,Z 170,A -170.5157,B 9.2165,C 0.274,E1 9.0619,E2 262.0712} C_DIS
Enddeposition()
END
